(* IEC 61131-3 sources: SmartHomeNew/ (part 10) *)

(* ---- FB_Water_Valve_Runtime_Governance.st ---- *)
FUNCTION_BLOCK FB_Water_Valve_Runtime_Governance
VAR_INPUT
    VI_Enable : BOOL;
    VI_System_Time_MS : UDINT;
END_VAR
VAR
    L_i : INT;
    L_Group : INT;
    L_Feedback_Index_A : INT;
    L_Feedback_Index_B : INT;

    L_Authority : ST_Water_Isolation_Authority_State;
    L_Valve : ST_Water_Valve_Runtime_State;
    L_Empty_Valve : ST_Water_Valve_Runtime_State;

    L_Feedback_A : ST_Water_Valve_Feedback_State;
    L_Feedback_B : ST_Water_Valve_Feedback_State;

    L_Any_Degraded : BOOL;
    L_Any_Confirmation_Unknown : BOOL;
    L_Any_Unsafe_Reopen : BOOL;
END_VAR

IF NOT VI_Enable THEN
    GVL_Water_Valve_Runtime.G_Runtime_Valid := FALSE;
    RETURN;
END_IF;

L_Any_Degraded := FALSE;
L_Any_Confirmation_Unknown := FALSE;
L_Any_Unsafe_Reopen := FALSE;

FOR L_i := 1 TO GVL_CONSTANTS.C_MAX_FLOOD_SENSORS DO

    L_Authority :=
        GVL_Water_Isolation_Authority.G_Authority_State[L_i];

    L_Valve := L_Empty_Valve;
    L_Valve.Runtime_Valid := TRUE;

    L_Valve.Runtime_System_Time_MS := VI_System_Time_MS;

    L_Valve.Valve_Id := L_Authority.Valve_Group_Id;
    L_Valve.Valve_Group_Id := L_Authority.Valve_Group_Id;

    L_Valve.Close_Requested :=
        L_Authority.Selective_Authority_Allowed
        OR L_Authority.Global_Fallback_Required;

    L_Valve.Global_Fallback_Request :=
        L_Authority.Global_Fallback_Required;

    L_Valve.Selective_Authority_Allowed :=
        L_Authority.Selective_Authority_Allowed;

    // Observe-only compatibility visibility.
    L_Valve.Physical_Output_Active :=
        GVL_COMMAND_SHADOW.G_Close_Valve_35
        OR GVL_COMMAND_SHADOW.G_Close_Valve_36;

    L_Valve.Output_Command_Projected :=
        L_Valve.Close_Requested;

    // Feedback/runtime hooks. Runtime authority is per leak sensor, but valve
    // feedback is per physical valve pair: group 1 => 1/2, group 2 => 3/4,
    // group 3 => 5/6, group 4 => 7/8 (35/36).
    L_Group := UINT_TO_INT(L_Authority.Valve_Group_Id);
    L_Feedback_Index_A := 0;
    L_Feedback_Index_B := 0;

    CASE L_Group OF
        1:
            L_Feedback_Index_A := 1;
            L_Feedback_Index_B := 2;
        2:
            L_Feedback_Index_A := 3;
            L_Feedback_Index_B := 4;
        3:
            L_Feedback_Index_A := 5;
            L_Feedback_Index_B := 6;
        4:
            L_Feedback_Index_A := 7;
            L_Feedback_Index_B := 8;
    ELSE
            L_Feedback_Index_A := 0;
            L_Feedback_Index_B := 0;
    END_CASE;

    IF (L_Feedback_Index_A >= 1) AND (L_Feedback_Index_B >= 1) THEN
        L_Feedback_A := GVL_Water_Valve_Feedback.G_Valve_Feedback_State[L_Feedback_Index_A];
        L_Feedback_B := GVL_Water_Valve_Feedback.G_Valve_Feedback_State[L_Feedback_Index_B];

        L_Valve.Confirmation_Available :=
            L_Feedback_A.Feedback_Available
            AND L_Feedback_B.Feedback_Available;

        IF L_Valve.Confirmation_Available THEN
            L_Valve.Confirmed_Closed :=
                L_Feedback_A.Confirmed_Closed
                AND L_Feedback_B.Confirmed_Closed;

            L_Valve.Confirmed_Open :=
                L_Feedback_A.Confirmed_Open
                AND L_Feedback_B.Confirmed_Open;

            L_Valve.Confirmation_Timeout :=
                L_Feedback_A.Feedback_Timeout
                OR L_Feedback_B.Feedback_Timeout;
        ELSE
            L_Valve.Confirmation_Unknown := TRUE;
        END_IF;
    ELSE
        L_Valve.Confirmation_Unknown := TRUE;
    END_IF;

    IF L_Valve.Confirmation_Available
       AND NOT L_Valve.Confirmed_Open
       AND NOT L_Valve.Confirmed_Closed THEN
        L_Valve.Confirmation_Unknown := TRUE;
    END_IF;

    // Observe-only semantics must not force degraded state.
    L_Valve.Diagnostics_Available := FALSE;
    L_Valve.Valve_Healthy := TRUE;

    IF L_Valve.Confirmation_Available
       AND NOT L_Valve.Confirmed_Closed
       AND L_Valve.Close_Requested THEN

        L_Valve.Valve_Degraded := TRUE;

    END_IF;

    IF L_Valve.Confirmation_Timeout THEN
        L_Valve.Valve_Degraded := TRUE;
        L_Valve.Valve_Stuck_Suspected := TRUE;
    END_IF;

    IF L_Valve.Valve_Degraded THEN

        L_Valve.Unsafe_Reopen_Denied := TRUE;
        L_Valve.Recovery_Allowed := FALSE;

        L_Valve.Status_Code := 2;
        L_Valve.Status_Text :=
            'Recovery denied: valve pair degraded';

    ELSIF L_Valve.Confirmation_Unknown THEN

        L_Valve.Status_Code := 1;
        L_Valve.Status_Text :=
            'Valve pair confirmation unavailable';

    ELSE

        L_Valve.Status_Code := 0;
        L_Valve.Status_Text :=
            'Valve pair governance runtime healthy';

    END_IF;

    GVL_Water_Valve_Runtime.G_Valve_Runtime_State[L_i] :=
        L_Valve;

    L_Any_Degraded :=
        L_Any_Degraded
        OR L_Valve.Valve_Degraded;

    L_Any_Confirmation_Unknown :=
        L_Any_Confirmation_Unknown
        OR L_Valve.Confirmation_Unknown;

    L_Any_Unsafe_Reopen :=
        L_Any_Unsafe_Reopen
        OR L_Valve.Unsafe_Reopen_Denied;

END_FOR;

GVL_Water_Valve_Runtime.G_Any_Valve_Degraded :=
    L_Any_Degraded;

GVL_Water_Valve_Runtime.G_Any_Confirmation_Unknown :=
    L_Any_Confirmation_Unknown;

GVL_Water_Valve_Runtime.G_Any_Unsafe_Reopen_Denied :=
    L_Any_Unsafe_Reopen;

GVL_Water_Valve_Runtime.G_Runtime_Valid := TRUE;
GVL_Water_Valve_Runtime.G_Last_Update_MS := VI_System_Time_MS;

IF L_Any_Degraded THEN
    GVL_Water_Valve_Runtime.G_Status_Code := 2;
    GVL_Water_Valve_Runtime.G_Status_Text :=
        'Valve governance degraded';
ELSIF L_Any_Confirmation_Unknown THEN
    GVL_Water_Valve_Runtime.G_Status_Code := 1;
    GVL_Water_Valve_Runtime.G_Status_Text :=
        'Valve pair confirmation unknown';
ELSE
    GVL_Water_Valve_Runtime.G_Status_Code := 0;
    GVL_Water_Valve_Runtime.G_Status_Text :=
        'Valve governance runtime active';
END_IF;

END_FUNCTION_BLOCK

(* ---- FB_Zone_Access_Manager.st ---- *)
FUNCTION_BLOCK FB_Zone_Access_Manager
VAR_INPUT
    VI_System_Time_MS : UDINT; // Системное время (мс)
    VI_Operator_ID    : STRING(10); // Идентификатор оператора
    VI_Target_Zone    : INT; // Номер целевой зоны
    VI_Rights         : ST_Operator_Zone_Rights; // Права доступа оператора к зоне
END_VAR
VAR_OUTPUT
    VO_Access_Granted : BOOL; // Флаг: Доступ разрешен
END_VAR

// Проверка прав доступа к зоне
IF VI_Target_Zone >= 1 AND VI_Target_Zone <= 32 THEN
    // Если глобальный уровень доступа высокий (например, CONFIG или FULL), разрешаем доступ ко всем зонам
    IF VI_Rights.global_access_level >= TO_BYTE(E_Zone_Access_Level.ZONE_ACCESS_CONFIG) THEN
        VO_Access_Granted := TRUE;
    ELSE
        // Иначе проверяем битовую маску для конкретной зоны
        // Бит 0 соответствует зоне 1, бит 1 - зоне 2 и т.д.
        VO_Access_Granted := (VI_Rights.zone_masks AND SHL(DWORD#1, VI_Target_Zone - 1)) <> 0;
    END_IF;
ELSE
    VO_Access_Granted := FALSE;
END_IF;

(* ---- MAIN.st ---- *)
PROGRAM MAIN

// ======================================================
// MAIN CYCLIC EXECUTION PIPELINE
// ======================================================
// Required CODESYS Task Configuration:
//   - Assign only PROGRAM MAIN to the cyclic task.
//   - Do not assign child PRG_* programs directly to the same task.
//   - Configure the real cycle time in CODESYS Task Configuration.
//   - Recommended main control cycle: 100 ms.
// ======================================================

// 1. Time / init / configuration
PRG_Time_Service();
PRG_Time_Monotonic_Governor();
PRG_System_Init();
PRG_Config_Manager();
PRG_Config_Validation();
PRG_Config_Versioning();
PRG_System_Runtime_Base();

// 2. Peer heartbeat ingestion
PRG_Peer_Heartbeat_Ingestion();

// 3. PLC role arbitration
PRG_PLC_Arbitration();

// 4. PLC ownership / fencing governance
PRG_PLC_Fencing_Governor();

// 5. IO read, passive quality observation and normalized inputs
PRG_IO_Read();
PRG_Input_Quality_Read();
PRG_Input_Processing();

// 6. Base mode, presence and safety
PRG_Mode_Manager();
PRG_Presence_Manager();
PRG_Safety();
PRG_Safety_Operator();
PRG_Safety_Shutdown();
PRG_Safety_Recovery();

// 7. Intent, adaptive behavior, scenario and policy
PRG_System_Intent();
PRG_Security();
PRG_System_Access_Maintenance();
PRG_User_Adapt_Control();
PRG_Behavior_Adapt_Profile();
PRG_Scenario_Engine();
PRG_System_Scenario_Rules();
PRG_System_Evacuation();
PRG_Policy();
PRG_Heating_Policy_Manager();
PRG_Heating_Policy_Observer();
PRG_System_Coordinator();

// 8. Command arbitration
PRG_Command_Arbitration();

// 9. Transport pipeline
PRG_Modbus_Master();
PRG_Modbus_RTU_Bridge();
PRG_Modbus_RTU_Driver();
PRG_Modbus_RTU_SysCom_Backend();
PRG_Modbus_RTU_SysCom_Transport();
PRG_Modbus_Register_Scan();
PRG_OpenTherm_Transport();
PRG_OpenTherm_Adapter_Status();

// 10. Transport freshness governance
PRG_Transport_Freshness_Governor();

// 11. Runtime authority barrier
PRG_Runtime_Barrier();

// 12. Immutable runtime snapshot governance
PRG_Runtime_Snapshot_Governor();

// 13. Canonical peer session publication
PRG_Peer_Session_Publication();

// 14. HA session replication boundary
PRG_HA_Session_Replication();

// 15. Distributed peer ingestion
PRG_Distributed_Peer_Ingestion();

// 16. Distributed epoch reconciliation governance
PRG_Distributed_Epoch_Governor();

// 17. Distributed snapshot publication
PRG_Distributed_Snapshot_Publication();

// 18. Distributed snapshot ingestion
PRG_Distributed_Snapshot_Ingestion();

// 19. Distributed immutable snapshot reconciliation governance
PRG_Distributed_Snapshot_Governor();

// 20. Distributed runtime fabric supervisor
PRG_Distributed_Runtime_Supervisor();

// 21. Distributed commit publication
PRG_Distributed_Commit_Publication();

// 22. Distributed commit ingestion
PRG_Distributed_Commit_Ingestion();

// 23. Distributed deterministic publication commit governance
PRG_Distributed_Commit_Governor();

// 24. Distributed deterministic commit observability projection
PRG_Distributed_Commit_Observability();

// 25. Semantic execution continuity governance
PRG_Semantic_Progress_Governor();

// 26. Systemic convergence governance
PRG_Convergence_Governor();

// 27. Recovery cleanup governance
PRG_Recovery_Cleanup_Governor();

// 28. Observability authority governance
PRG_Observability_Governor();

// 29. Domain execution and projection
PRG_Heating();
PRG_Heating_Supervisory_Publication();
PRG_Ventilation();
PRG_Water_Supervisory_Publication();
PRG_Water_Output_Projection();
PRG_Water();
PRG_Access();
PRG_Lighting();

// 30. Output freshness governance
PRG_Output_Freshness_Governor();

// 31. Immutable physical snapshot governance
PRG_Physical_Snapshot_Governor();

// 32. Physical sensor consensus governance
PRG_Sensor_Consensus_Governor();

// 33. Telemetry causality governance
PRG_Telemetry_Causality_Governor();

// 34. Global physical authority epoch governance
PRG_Physical_Authority_Epoch_Governor();

// 35. Persistent authority lineage governance
PRG_Authority_Lineage_Governor();

// 36. Global authority revocation governance
PRG_Authority_Revocation_Governor();

// 37. Deterministic authority restoration governance
PRG_Authority_Restoration_Governor();

// 38. Pre-output safety barrier
PRG_PreOutput_Safety_Barrier();

// 39. Final physical IO projection
PRG_IO_Write();

// 40. Deterministic field actuation governance
PRG_Actuation_Authority_Governor();

// 41. Deterministic physical transaction governance
PRG_Physical_Transaction_Governor();

// 42. Deterministic temporal stability governance
PRG_Temporal_Stability_Governor();

// 43. Environmental authority governance
PRG_Environmental_Authority_Governor();

// 44. Runtime resource authority governance
PRG_Runtime_Resource_Authority_Governor();

// 45. Semantic continuity authority governance
PRG_Semantic_Continuity_Authority_Governor();

// 46. Authoritative observability truth governance
PRG_Observability_Truth_Governor();

// 47. Immutable historical truth governance
PRG_Historical_Truth_Governor();

// 48. Global synchronized authority governance
PRG_Global_Authority_Sync_Governor();

// 49. Deterministic control temporal coherence governance
PRG_Control_Temporal_Coherence_Governor();

// 50. Physical actuator semantic verification governance
PRG_Actuator_Semantic_Verification_Governor();

// 51. Deterministic energy causality governance
PRG_Energy_Causality_Governor();

// 52. Deterministic runtime sustainability governance
PRG_Runtime_Sustainability_Governor();

// 53. Deterministic semantic preservation governance
PRG_Semantic_Preservation_Governor();

// 54. Deterministic operator semantic alignment governance
PRG_Operator_Semantic_Alignment_Governor();

// 55. Deterministic ecosystem semantic federation governance
PRG_Semantic_Federation_Governor();

// 56. Deterministic compliance federation governance
PRG_Compliance_Federation_Governor();

// 57. Deterministic forensic evidence governance
PRG_Forensic_Evidence_Governor();

// 58. Deterministic epistemic integrity governance
PRG_Epistemic_Integrity_Governor();

// 59. Deterministic meta-governance consistency governance
// Must run before observability authority publication to guarantee
// acyclic and independently grounded governance topology.
PRG_Meta_Governance_Governor();

// 60. Observability authority coherence governance
PRG_Observability_Authority_Governor();

// 61. Verification, diagnostics, history, HMI
PRG_Command_Verifier();
PRG_Explainability();
PRG_System_Health();
PRG_System_Alarm_Gateway();
PRG_System_Diagnostics();
PRG_System_Diagnostics_Ext();
PRG_System_History();
PRG_System_BlackBox();
PRG_System_Trend();
PRG_System_Simulation();
PRG_HMI_Dashboard();
PRG_Debug_View();

// >>> BULK_SYNC_ANCHOR: MAIN <<<
END_PROGRAM

(* ---- PRG_Access.st ---- *)
PROGRAM PRG_Access
VAR
    fbProjection : FB_Access_Output_Projection;

    fbPulseLock1Open : FB_Access_Pulse_Channel;
    fbPulseLock1Close : FB_Access_Pulse_Channel;
    fbPulseLock2Open : FB_Access_Pulse_Channel;
    fbPulseLock2Close : FB_Access_Pulse_Channel;
    fbPulseGateOpen : FB_Access_Pulse_Channel;
    fbPulseWicketOpen : FB_Access_Pulse_Channel;

    L_Mode : E_Safety_Mode;
    L_Now_MS : UDINT;
    L_Pulse_MS : UDINT;

    L_Distributed_Execute_Allowed : BOOL;
    L_Distributed_Access_Allowed : BOOL;

    L_Lock_1_Open : BOOL;
    L_Lock_1_Close : BOOL;
    L_Lock_2_Open : BOOL;
    L_Lock_2_Close : BOOL;
    L_Gate_Open : BOOL;
    L_Wicket_Open : BOOL;
END_VAR

L_Mode := GVL_SAFETY_SHUTDOWN.G_Safety_Mode;
L_Now_MS := GVL_STATUS.G_System_Time_MS;

GVL_ACCESS_RUNTIME.G_Runtime_Required := FALSE;
GVL_ACCESS_RUNTIME.G_Runtime_Executed := TRUE;
GVL_ACCESS_RUNTIME.G_Runtime_Idle_By_Design := FALSE;
GVL_ACCESS_RUNTIME.G_Runtime_Blocked_By_Distributed_Gates := FALSE;
GVL_ACCESS_RUNTIME.G_Any_Pulse_Active := FALSE;
GVL_ACCESS_RUNTIME.G_Last_Update_MS := L_Now_MS;

// Distributed runtime governance.
// FIRE/GAS emergency semantics remain authoritative.
L_Distributed_Execute_Allowed :=
    GVL_Distributed_Execution_Gates.G_Can_Execute;

L_Distributed_Access_Allowed :=
    GVL_Distributed_Execution_Gates.G_Can_Own_Projection;

IF (L_Mode <> FIRE)
   AND (L_Mode <> GAS)
   AND (
        NOT L_Distributed_Execute_Allowed
        OR NOT L_Distributed_Access_Allowed
       ) THEN

    // Clear all pulse channels before blocking projection to avoid stale pulse-active state.
    fbPulseLock1Open(VI_Command := FALSE, VI_Reset := TRUE, VI_Now_MS := L_Now_MS, VI_Pulse_MS := 100);
    fbPulseLock1Close(VI_Command := FALSE, VI_Reset := TRUE, VI_Now_MS := L_Now_MS, VI_Pulse_MS := 100);
    fbPulseLock2Open(VI_Command := FALSE, VI_Reset := TRUE, VI_Now_MS := L_Now_MS, VI_Pulse_MS := 100);
    fbPulseLock2Close(VI_Command := FALSE, VI_Reset := TRUE, VI_Now_MS := L_Now_MS, VI_Pulse_MS := 100);
    fbPulseGateOpen(VI_Command := FALSE, VI_Reset := TRUE, VI_Now_MS := L_Now_MS, VI_Pulse_MS := 100);
    fbPulseWicketOpen(VI_Command := FALSE, VI_Reset := TRUE, VI_Now_MS := L_Now_MS, VI_Pulse_MS := 100);

    fbProjection(
        VI_Lock_1_Open := FALSE,
        VI_Lock_1_Close := FALSE,
        VI_Lock_2_Open := FALSE,
        VI_Lock_2_Close := FALSE,
        VI_Gate_Open := FALSE,
        VI_Wicket_Open := FALSE
    );

    GVL_ACCESS_RUNTIME.G_Runtime_Blocked_By_Distributed_Gates := TRUE;
    GVL_ACCESS_RUNTIME.G_Any_Pulse_Active := FALSE;
    GVL_ACCESS_RUNTIME.G_Status_Code := 2;
    GVL_ACCESS_RUNTIME.G_Status_Text := 'Access runtime blocked by distributed gates';

    RETURN;
END_IF;

// Access is not part of WATER_LEAK or GLOBAL_STOP recovery semantics.
// Clear active one-shot pulses so old manual commands cannot continue during safety stop.
IF (L_Mode = WATER_LEAK) OR (L_Mode = GLOBAL_STOP) THEN
    fbPulseLock1Open(VI_Command := FALSE, VI_Reset := TRUE, VI_Now_MS := L_Now_MS, VI_Pulse_MS := 100);
    fbPulseLock1Close(VI_Command := FALSE, VI_Reset := TRUE, VI_Now_MS := L_Now_MS, VI_Pulse_MS := 100);
    fbPulseLock2Open(VI_Command := FALSE, VI_Reset := TRUE, VI_Now_MS := L_Now_MS, VI_Pulse_MS := 100);
    fbPulseLock2Close(VI_Command := FALSE, VI_Reset := TRUE, VI_Now_MS := L_Now_MS, VI_Pulse_MS := 100);
    fbPulseGateOpen(VI_Command := FALSE, VI_Reset := TRUE, VI_Now_MS := L_Now_MS, VI_Pulse_MS := 100);
    fbPulseWicketOpen(VI_Command := FALSE, VI_Reset := TRUE, VI_Now_MS := L_Now_MS, VI_Pulse_MS := 100);

    fbProjection(
        VI_Lock_1_Open := FALSE,
        VI_Lock_1_Close := FALSE,
        VI_Lock_2_Open := FALSE,
        VI_Lock_2_Close := FALSE,
        VI_Gate_Open := FALSE,
        VI_Wicket_Open := FALSE
    );

    GVL_ACCESS_RUNTIME.G_Runtime_Required := FALSE;
    GVL_ACCESS_RUNTIME.G_Runtime_Idle_By_Design := TRUE;
    GVL_ACCESS_RUNTIME.G_Any_Pulse_Active := FALSE;
    GVL_ACCESS_RUNTIME.G_Status_Code := 3;
    GVL_ACCESS_RUNTIME.G_Status_Text := 'Access runtime safety-cleared';

    RETURN;
END_IF;

// Load pulse duration from config with safety clamp.
L_Pulse_MS := GVL_CONFIG.G_Access_Pulse_MS;
IF L_Pulse_MS < 100 THEN
    L_Pulse_MS := 100;
ELSIF L_Pulse_MS > 5000 THEN
    L_Pulse_MS := 5000;
END_IF;

L_Lock_1_Open := FALSE;
L_Lock_1_Close := FALSE;
L_Lock_2_Open := FALSE;
L_Lock_2_Close := FALSE;
L_Gate_Open := FALSE;
L_Wicket_Open := FALSE;

CASE L_Mode OF
    FIRE:
        // Fire evacuation access commands are authoritative and continuous.
        L_Lock_1_Open := GVL_COMMAND_SHADOW.G_Lock_1_Open;
        L_Lock_2_Open := GVL_COMMAND_SHADOW.G_Lock_2_Open;
        L_Gate_Open := GVL_COMMAND_SHADOW.G_Gate_Open;
        L_Wicket_Open := GVL_COMMAND_SHADOW.G_Wicket_Open;

        // Synchronize pulse channels with current command state and clear active pulses.
        fbPulseLock1Open(VI_Command := GVL_COMMAND_SHADOW.G_Lock_1_Open, VI_Reset := TRUE, VI_Now_MS := L_Now_MS, VI_Pulse_MS := L_Pulse_MS);
        fbPulseLock1Close(VI_Command := GVL_COMMAND_SHADOW.G_Lock_1_Close, VI_Reset := TRUE, VI_Now_MS := L_Now_MS, VI_Pulse_MS := L_Pulse_MS);
        fbPulseLock2Open(VI_Command := GVL_COMMAND_SHADOW.G_Lock_2_Open, VI_Reset := TRUE, VI_Now_MS := L_Now_MS, VI_Pulse_MS := L_Pulse_MS);
        fbPulseLock2Close(VI_Command := GVL_COMMAND_SHADOW.G_Lock_2_Close, VI_Reset := TRUE, VI_Now_MS := L_Now_MS, VI_Pulse_MS := L_Pulse_MS);
        fbPulseGateOpen(VI_Command := GVL_COMMAND_SHADOW.G_Gate_Open, VI_Reset := TRUE, VI_Now_MS := L_Now_MS, VI_Pulse_MS := L_Pulse_MS);
        fbPulseWicketOpen(VI_Command := GVL_COMMAND_SHADOW.G_Wicket_Open, VI_Reset := TRUE, VI_Now_MS := L_Now_MS, VI_Pulse_MS := L_Pulse_MS);

    GAS:
        // Gas mode uses direct gate opening plus limited pulsed pedestrian/lock release.
        L_Gate_Open := GVL_COMMAND_SHADOW.G_Gate_Open;

        fbPulseLock1Open(VI_Command := GVL_COMMAND_SHADOW.G_Lock_1_Open, VI_Reset := FALSE, VI_Now_MS := L_Now_MS, VI_Pulse_MS := L_Pulse_MS);
        fbPulseLock2Open(VI_Command := GVL_COMMAND_SHADOW.G_Lock_2_Open, VI_Reset := FALSE, VI_Now_MS := L_Now_MS, VI_Pulse_MS := L_Pulse_MS);
        fbPulseWicketOpen(VI_Command := GVL_COMMAND_SHADOW.G_Wicket_Open, VI_Reset := FALSE, VI_Now_MS := L_Now_MS, VI_Pulse_MS := L_Pulse_MS);

        fbPulseLock1Close(VI_Command := GVL_COMMAND_SHADOW.G_Lock_1_Close, VI_Reset := TRUE, VI_Now_MS := L_Now_MS, VI_Pulse_MS := L_Pulse_MS);
        fbPulseLock2Close(VI_Command := GVL_COMMAND_SHADOW.G_Lock_2_Close, VI_Reset := TRUE, VI_Now_MS := L_Now_MS, VI_Pulse_MS := L_Pulse_MS);
        fbPulseGateOpen(VI_Command := GVL_COMMAND_SHADOW.G_Gate_Open, VI_Reset := TRUE, VI_Now_MS := L_Now_MS, VI_Pulse_MS := L_Pulse_MS);

        L_Lock_1_Open := fbPulseLock1Open.VO_Output;
        L_Lock_2_Open := fbPulseLock2Open.VO_Output;
        L_Wicket_Open := fbPulseWicketOpen.VO_Output;

ELSE
        fbPulseLock1Open(VI_Command := GVL_COMMAND_SHADOW.G_Lock_1_Open, VI_Reset := FALSE, VI_Now_MS := L_Now_MS, VI_Pulse_MS := L_Pulse_MS);
        fbPulseLock1Close(VI_Command := GVL_COMMAND_SHADOW.G_Lock_1_Close, VI_Reset := FALSE, VI_Now_MS := L_Now_MS, VI_Pulse_MS := L_Pulse_MS);
        fbPulseLock2Open(VI_Command := GVL_COMMAND_SHADOW.G_Lock_2_Open, VI_Reset := FALSE, VI_Now_MS := L_Now_MS, VI_Pulse_MS := L_Pulse_MS);
        fbPulseLock2Close(VI_Command := GVL_COMMAND_SHADOW.G_Lock_2_Close, VI_Reset := FALSE, VI_Now_MS := L_Now_MS, VI_Pulse_MS := L_Pulse_MS);
        fbPulseGateOpen(VI_Command := GVL_COMMAND_SHADOW.G_Gate_Open, VI_Reset := FALSE, VI_Now_MS := L_Now_MS, VI_Pulse_MS := L_Pulse_MS);
        fbPulseWicketOpen(VI_Command := GVL_COMMAND_SHADOW.G_Wicket_Open, VI_Reset := FALSE, VI_Now_MS := L_Now_MS, VI_Pulse_MS := L_Pulse_MS);

        L_Lock_1_Open := fbPulseLock1Open.VO_Output;
        L_Lock_1_Close := fbPulseLock1Close.VO_Output;
        L_Lock_2_Open := fbPulseLock2Open.VO_Output;
        L_Lock_2_Close := fbPulseLock2Close.VO_Output;
        L_Gate_Open := fbPulseGateOpen.VO_Output;
        L_Wicket_Open := fbPulseWicketOpen.VO_Output;
END_CASE;

GVL_ACCESS_RUNTIME.G_Any_Pulse_Active :=
    fbPulseLock1Open.VO_Active
    OR fbPulseLock1Close.VO_Active
    OR fbPulseLock2Open.VO_Active
    OR fbPulseLock2Close.VO_Active
    OR fbPulseGateOpen.VO_Active
    OR fbPulseWicketOpen.VO_Active;

GVL_ACCESS_RUNTIME.G_Runtime_Required :=
    (L_Mode = FIRE)
    OR (L_Mode = GAS)
    OR GVL_COMMAND_SHADOW.G_Lock_1_Open
    OR GVL_COMMAND_SHADOW.G_Lock_1_Close
    OR GVL_COMMAND_SHADOW.G_Lock_2_Open
    OR GVL_COMMAND_SHADOW.G_Lock_2_Close
    OR GVL_COMMAND_SHADOW.G_Gate_Open
    OR GVL_COMMAND_SHADOW.G_Wicket_Open
    OR GVL_ACCESS_RUNTIME.G_Any_Pulse_Active;

GVL_ACCESS_RUNTIME.G_Runtime_Idle_By_Design :=
    NOT GVL_ACCESS_RUNTIME.G_Runtime_Required;

IF GVL_ACCESS_RUNTIME.G_Runtime_Idle_By_Design THEN
    GVL_ACCESS_RUNTIME.G_Status_Code := 0;
    GVL_ACCESS_RUNTIME.G_Status_Text := 'Access runtime idle by design';
ELSE
    GVL_ACCESS_RUNTIME.G_Status_Code := 1;
    GVL_ACCESS_RUNTIME.G_Status_Text := 'Access runtime active';
END_IF;

fbProjection(
    VI_Lock_1_Open := L_Lock_1_Open,
    VI_Lock_1_Close := L_Lock_1_Close,
    VI_Lock_2_Open := L_Lock_2_Open,
    VI_Lock_2_Close := L_Lock_2_Close,
    VI_Gate_Open := L_Gate_Open,
    VI_Wicket_Open := L_Wicket_Open
);

// >>> BULK_SYNC_ANCHOR: PRG_Access <<<
END_PROGRAM

(* ---- PRG_Actuation_Authority_Governor.st ---- *)
PROGRAM PRG_Actuation_Authority_Governor
VAR
    L_Now_MS : UDINT;
    L_Actuation_Valid : BOOL := TRUE;
    L_Error_Code : UDINT := 0;
    L_Error_Text : STRING(160) := '';
END_VAR

L_Now_MS := GVL_STATUS.G_System_Time_MS;
L_Actuation_Valid := TRUE;
L_Error_Code := 0;
L_Error_Text := '';

GVL_ACTUATION_AUTHORITY.Actuation_Authority_Valid := FALSE;
GVL_ACTUATION_AUTHORITY.Actuation_Authority_Granted := FALSE;
GVL_ACTUATION_AUTHORITY.Actuation_Quarantine_Active := TRUE;
GVL_ACTUATION_AUTHORITY.Field_Device_ACK_Valid := FALSE;
GVL_ACTUATION_AUTHORITY.Actuator_Transition_Observed := FALSE;
GVL_ACTUATION_AUTHORITY.Physical_Convergence_Confirmed := FALSE;
GVL_ACTUATION_AUTHORITY.Stable_Physical_Convergence := FALSE;

GVL_ACTUATION_AUTHORITY.Actuation_Command_Epoch := ULINT_TO_UDINT(GVL_OUTPUT_EPOCH.Output_Publication_Epoch);

IF GVL_ACTUATION_AUTHORITY.Field_ACK_Epoch <> GVL_ACTUATION_AUTHORITY.Actuation_Command_Epoch THEN
    GVL_ACTUATION_AUTHORITY.Command_Actuation_Skew_Detected := TRUE;
    L_Actuation_Valid := FALSE;
    L_Error_Code := 26000;
    L_Error_Text := 'Command actuation epoch skew detected';
END_IF;

IF L_Actuation_Valid AND GVL_ACTUATION_AUTHORITY.ACK_Replay_Suspected THEN
    L_Actuation_Valid := FALSE;
    L_Error_Code := 26001;
    L_Error_Text := 'Field ACK replay suspected';
END_IF;

IF L_Actuation_Valid AND GVL_ACTUATION_AUTHORITY.Write_Without_Confirm_Detected THEN
    L_Actuation_Valid := FALSE;
    L_Error_Code := 26002;
    L_Error_Text := 'Write without field confirmation detected';
END_IF;

IF L_Actuation_Valid AND GVL_ACTUATION_AUTHORITY.Relay_Weld_Suspected THEN
    L_Actuation_Valid := FALSE;
    L_Error_Code := 26003;
    L_Error_Text := 'Relay weld suspected';
END_IF;

IF L_Actuation_Valid AND GVL_ACTUATION_AUTHORITY.Actuator_Stall_Detected THEN
    L_Actuation_Valid := FALSE;
    L_Error_Code := 26004;
    L_Error_Text := 'Actuator stall detected';
END_IF;

IF L_Actuation_Valid AND GVL_ACTUATION_AUTHORITY.Partial_Actuation_Detected THEN
    L_Actuation_Valid := FALSE;
    L_Error_Code := 26005;
    L_Error_Text := 'Partial actuation detected';
END_IF;

IF L_Actuation_Valid AND NOT GVL_ACTUATION_AUTHORITY.Current_Signature_Confirmed THEN
    L_Actuation_Valid := FALSE;
    L_Error_Code := 26010;
    L_Error_Text := 'Current signature confirmation missing';
END_IF;

IF L_Actuation_Valid AND NOT GVL_ACTUATION_AUTHORITY.Flow_Response_Confirmed THEN
    L_Actuation_Valid := FALSE;
    L_Error_Code := 26011;
    L_Error_Text := 'Flow response confirmation missing';
END_IF;

IF L_Actuation_Valid AND NOT GVL_ACTUATION_AUTHORITY.Pressure_Response_Confirmed THEN
    L_Actuation_Valid := FALSE;
    L_Error_Code := 26012;
    L_Error_Text := 'Pressure response confirmation missing';
END_IF;

IF L_Actuation_Valid AND NOT GVL_ACTUATION_AUTHORITY.Motion_Response_Confirmed THEN
    L_Actuation_Valid := FALSE;
    L_Error_Code := 26013;
    L_Error_Text := 'Motion response confirmation missing';
END_IF;

IF L_Actuation_Valid THEN
    GVL_ACTUATION_AUTHORITY.Actuation_Authority_Valid := TRUE;
    GVL_ACTUATION_AUTHORITY.Actuation_Authority_Granted := TRUE;
    GVL_ACTUATION_AUTHORITY.Actuation_Quarantine_Active := FALSE;
    GVL_ACTUATION_AUTHORITY.Field_Device_ACK_Valid := TRUE;
    GVL_ACTUATION_AUTHORITY.Actuator_Transition_Observed := TRUE;
    GVL_ACTUATION_AUTHORITY.Physical_Convergence_Confirmed := TRUE;
    GVL_ACTUATION_AUTHORITY.Stable_Physical_Convergence := TRUE;
    GVL_ACTUATION_AUTHORITY.Actuation_Authority_Epoch := GVL_ACTUATION_AUTHORITY.Actuation_Command_Epoch;
    GVL_ACTUATION_AUTHORITY.Actuation_Last_Update_MS := L_Now_MS;
    GVL_ACTUATION_AUTHORITY.Actuation_Lease_Expired := FALSE;
    GVL_ACTUATION_AUTHORITY.Actuation_Last_Error_Code := 0;
    GVL_ACTUATION_AUTHORITY.Actuation_Last_Error_Text := '';
ELSE
    GVL_ACTUATION_AUTHORITY.Actuation_Authority_Valid := FALSE;
    GVL_ACTUATION_AUTHORITY.Actuation_Authority_Granted := FALSE;
    GVL_ACTUATION_AUTHORITY.Actuation_Quarantine_Active := TRUE;
    GVL_ACTUATION_AUTHORITY.Actuation_Lease_Expired := TRUE;
    GVL_ACTUATION_AUTHORITY.Actuation_Last_Error_Code := L_Error_Code;
    GVL_ACTUATION_AUTHORITY.Actuation_Last_Error_Text := L_Error_Text;
    GVL_ACTUATION_AUTHORITY.Actuation_Invalidation_Count := GVL_ACTUATION_AUTHORITY.Actuation_Invalidation_Count + 1;
END_IF;

END_PROGRAM

(* ---- PRG_Actuator_Semantic_Verification_Governor.st ---- *)
PROGRAM PRG_Actuator_Semantic_Verification_Governor
VAR
    L_Now_MS : UDINT;
    L_Actuator_Valid : BOOL := TRUE;
    L_Error_Code : UDINT := 0;
    L_Error_Text : STRING(160) := '';
END_VAR

L_Now_MS := GVL_STATUS.G_System_Time_MS;
L_Actuator_Valid := TRUE;
L_Error_Code := 0;
L_Error_Text := '';

// Fail-safe defaults.
GVL_ACTUATOR_SEMANTIC_VERIFICATION.Actuator_Semantic_Verification_Valid := FALSE;
GVL_ACTUATOR_SEMANTIC_VERIFICATION.Actuator_Semantic_Verification_Granted := FALSE;
GVL_ACTUATOR_SEMANTIC_VERIFICATION.Actuator_Semantic_Verification_Quarantine_Active := TRUE;

GVL_ACTUATOR_SEMANTIC_VERIFICATION.Valve_Semantic_Realization_Valid := FALSE;
GVL_ACTUATOR_SEMANTIC_VERIFICATION.Relay_Semantic_Realization_Valid := FALSE;
GVL_ACTUATOR_SEMANTIC_VERIFICATION.Pump_Semantic_Realization_Valid := FALSE;
GVL_ACTUATOR_SEMANTIC_VERIFICATION.Fan_Semantic_Realization_Valid := FALSE;
GVL_ACTUATOR_SEMANTIC_VERIFICATION.Hydraulic_Response_Valid := FALSE;

// Control temporal coherence required.
IF NOT GVL_CONTROL_TIMING_FABRIC.Control_Temporal_Coherence_Granted THEN
    L_Actuator_Valid := FALSE;
    L_Error_Code := 36000;
    L_Error_Text := 'Control temporal coherence not granted';
END_IF;

// Semantic realization failure detectors.
IF GVL_ACTUATOR_SEMANTIC_VERIFICATION.False_Positive_Actuation_Detected THEN
    L_Actuator_Valid := FALSE;
    L_Error_Code := 36001;
    L_Error_Text := 'False-positive actuation detected';
END_IF;

IF GVL_ACTUATOR_SEMANTIC_VERIFICATION.Mechanical_NonRealization_Detected THEN
    L_Actuator_Valid := FALSE;
    L_Error_Code := 36002;
    L_Error_Text := 'Mechanical non-realization detected';
END_IF;

IF GVL_ACTUATOR_SEMANTIC_VERIFICATION.Welded_Relay_Semantics_Detected THEN
    L_Actuator_Valid := FALSE;
    L_Error_Code := 36003;
    L_Error_Text := 'Welded relay semantics detected';
END_IF;

IF GVL_ACTUATOR_SEMANTIC_VERIFICATION.Hydraulic_NoEffect_Execution_Detected THEN
    L_Actuator_Valid := FALSE;
    L_Error_Code := 36004;
    L_Error_Text := 'Hydraulic no-effect execution detected';
END_IF;

IF GVL_ACTUATOR_SEMANTIC_VERIFICATION.Airflow_Realization_Mismatch_Detected THEN
    L_Actuator_Valid := FALSE;
    L_Error_Code := 36005;
    L_Error_Text := 'Airflow realization mismatch detected';
END_IF;

IF GVL_ACTUATOR_SEMANTIC_VERIFICATION.Physical_Convergence_Divergence_Detected THEN
    L_Actuator_Valid := FALSE;
    L_Error_Code := 36006;
    L_Error_Text := 'Physical convergence divergence detected';
END_IF;

// Physical semantic convergence validation.
IF L_Actuator_Valid
AND NOT GVL_ACTUATOR_SEMANTIC_VERIFICATION.Physical_Effect_Converged THEN
    L_Actuator_Valid := FALSE;
    L_Error_Code := 36010;
    L_Error_Text := 'Physical effect convergence invalid';
END_IF;

IF L_Actuator_Valid
AND NOT GVL_ACTUATOR_SEMANTIC_VERIFICATION.Actuation_Response_Temporal_Valid THEN
    L_Actuator_Valid := FALSE;
    L_Error_Code := 36011;
    L_Error_Text := 'Actuation response timing invalid';
END_IF;

IF L_Actuator_Valid
AND NOT GVL_ACTUATOR_SEMANTIC_VERIFICATION.Sensor_Confirmed_Execution_Valid THEN
    L_Actuator_Valid := FALSE;
    L_Error_Code := 36012;
    L_Error_Text := 'Sensor-confirmed execution invalid';
END_IF;

IF L_Actuator_Valid
AND NOT GVL_ACTUATOR_SEMANTIC_VERIFICATION.Semantic_Outcome_Aligned THEN
    L_Actuator_Valid := FALSE;
    L_Error_Code := 36013;
    L_Error_Text := 'Semantic outcome alignment invalid';
END_IF;

IF L_Actuator_Valid THEN
    GVL_ACTUATOR_SEMANTIC_VERIFICATION.Actuator_Semantic_Verification_Valid := TRUE;
    GVL_ACTUATOR_SEMANTIC_VERIFICATION.Actuator_Semantic_Verification_Granted := TRUE;
    GVL_ACTUATOR_SEMANTIC_VERIFICATION.Actuator_Semantic_Verification_Quarantine_Active := FALSE;

    GVL_ACTUATOR_SEMANTIC_VERIFICATION.Valve_Semantic_Realization_Valid := TRUE;
    GVL_ACTUATOR_SEMANTIC_VERIFICATION.Relay_Semantic_Realization_Valid := TRUE;
    GVL_ACTUATOR_SEMANTIC_VERIFICATION.Pump_Semantic_Realization_Valid := TRUE;
    GVL_ACTUATOR_SEMANTIC_VERIFICATION.Fan_Semantic_Realization_Valid := TRUE;
    GVL_ACTUATOR_SEMANTIC_VERIFICATION.Hydraulic_Response_Valid := TRUE;

    GVL_ACTUATOR_SEMANTIC_VERIFICATION.Actuator_Verification_Epoch :=
        GVL_CONTROL_TIMING_FABRIC.Control_Timing_Epoch;

    GVL_ACTUATOR_SEMANTIC_VERIFICATION.Actuator_Verification_Epoch_Coherent := TRUE;

    GVL_ACTUATOR_SEMANTIC_VERIFICATION.Actuator_Verification_Last_Update_MS :=
        L_Now_MS;

    GVL_ACTUATOR_SEMANTIC_VERIFICATION.Actuator_Verification_Lease_Expired := FALSE;

    GVL_ACTUATOR_SEMANTIC_VERIFICATION.Actuator_Verification_Last_Error_Code := 0;
    GVL_ACTUATOR_SEMANTIC_VERIFICATION.Actuator_Verification_Last_Error_Text := '';
ELSE
    GVL_ACTUATOR_SEMANTIC_VERIFICATION.Actuator_Semantic_Verification_Valid := FALSE;
    GVL_ACTUATOR_SEMANTIC_VERIFICATION.Actuator_Semantic_Verification_Granted := FALSE;
    GVL_ACTUATOR_SEMANTIC_VERIFICATION.Actuator_Semantic_Verification_Quarantine_Active := TRUE;

    GVL_ACTUATOR_SEMANTIC_VERIFICATION.Actuator_Verification_Lease_Expired := TRUE;

    GVL_ACTUATOR_SEMANTIC_VERIFICATION.Actuator_Verification_Last_Error_Code :=
        L_Error_Code;

    GVL_ACTUATOR_SEMANTIC_VERIFICATION.Actuator_Verification_Last_Error_Text :=
        L_Error_Text;

    GVL_ACTUATOR_SEMANTIC_VERIFICATION.Actuator_Verification_Invalidation_Count :=
        GVL_ACTUATOR_SEMANTIC_VERIFICATION.Actuator_Verification_Invalidation_Count + 1;
END_IF;

END_PROGRAM

(* ---- PRG_Alarm_Audible_Ack_Manager.st ---- *)
PROGRAM PRG_Alarm_Audible_Ack_Manager
VAR
    L_Audible_Alarm_Active : BOOL;
    L_Remaining_MS : UDINT;
END_VAR

L_Audible_Alarm_Active := GVL_ALARM.G_Global_Critical OR GVL_ALARM.G_Gas_Fire_Siren OR GVL_ALARM.G_Security_Siren;
GVL_ALARM_AUDIBLE_ACK.G_Last_Ack_Accepted := FALSE;
GVL_ALARM_AUDIBLE_ACK.G_Last_Ack_Denied := FALSE;
GVL_ALARM_AUDIBLE_ACK.G_Last_Denial_Code := 0;

IF NOT L_Audible_Alarm_Active THEN
    GVL_ALARM_AUDIBLE_ACK.G_Ack_Active := FALSE;
    GVL_ALARM_AUDIBLE_ACK.G_Ack_Expires_MS := 0;
    GVL_ALARM_AUDIBLE_ACK.G_Ack_Remaining_MS := 0;
    GVL_ALARM_AUDIBLE_ACK.G_Ack_Count_Current_Alarm := 0;
    GVL_ALARM_AUDIBLE_ACK.G_Ack_Limit_Reached := FALSE;
    GVL_ALARM_AUDIBLE_ACK.G_Status_Text := 'Audible alarm acknowledgement idle';
END_IF;

IF GVL_ALARM_AUDIBLE_ACK.G_Ack_Active THEN
    IF GVL_TIME_SERVICE.G_Now_MS >= GVL_ALARM_AUDIBLE_ACK.G_Ack_Expires_MS THEN
        GVL_ALARM_AUDIBLE_ACK.G_Ack_Active := FALSE;
        GVL_ALARM_AUDIBLE_ACK.G_Ack_Remaining_MS := 0;
        GVL_ALARM_AUDIBLE_ACK.G_Status_Text := 'Audible alarm acknowledgement expired';
    ELSE
        L_Remaining_MS := GVL_ALARM_AUDIBLE_ACK.G_Ack_Expires_MS - GVL_TIME_SERVICE.G_Now_MS;
        GVL_ALARM_AUDIBLE_ACK.G_Ack_Remaining_MS := L_Remaining_MS;
    END_IF;
END_IF;

IF GVL_ALARM_AUDIBLE_ACK.G_Ack_Request THEN
    IF NOT L_Audible_Alarm_Active THEN
        GVL_ALARM_AUDIBLE_ACK.G_Last_Ack_Denied := TRUE;
        GVL_ALARM_AUDIBLE_ACK.G_Last_Denial_Code := 1;
        GVL_ALARM_AUDIBLE_ACK.G_Status_Text := 'Audible acknowledgement denied: no active audible alarm';
    ELSIF GVL_INTENT_USER.I_User_Access_Level < 2 THEN
        GVL_ALARM_AUDIBLE_ACK.G_Last_Ack_Denied := TRUE;
        GVL_ALARM_AUDIBLE_ACK.G_Last_Denial_Code := 2;
        GVL_ALARM_AUDIBLE_ACK.G_Status_Text := 'Audible acknowledgement denied: access level < 2';
    ELSIF GVL_ALARM_AUDIBLE_ACK.G_Ack_Count_Current_Alarm >= 3 THEN
        GVL_ALARM_AUDIBLE_ACK.G_Last_Ack_Denied := TRUE;
        GVL_ALARM_AUDIBLE_ACK.G_Last_Denial_Code := 3;
        GVL_ALARM_AUDIBLE_ACK.G_Ack_Limit_Reached := TRUE;
        GVL_ALARM_AUDIBLE_ACK.G_Status_Text := 'Audible acknowledgement denied: limit reached';
    ELSE
        GVL_ALARM_AUDIBLE_ACK.G_Ack_Count_Current_Alarm := GVL_ALARM_AUDIBLE_ACK.G_Ack_Count_Current_Alarm + 1;
        GVL_ALARM_AUDIBLE_ACK.G_Ack_Active := TRUE;
        GVL_ALARM_AUDIBLE_ACK.G_Ack_Expires_MS := GVL_TIME_SERVICE.G_Now_MS + (GVL_CONSTANTS.C_MS_IN_MINUTE * 5);
        GVL_ALARM_AUDIBLE_ACK.G_Ack_Remaining_MS := GVL_CONSTANTS.C_MS_IN_MINUTE * 5;
        GVL_ALARM_AUDIBLE_ACK.G_Last_Ack_Accepted := TRUE;
        GVL_ALARM_AUDIBLE_ACK.G_Last_Event_MS := GVL_TIME_SERVICE.G_Now_MS;
        GVL_ALARM_AUDIBLE_ACK.G_Status_Text := 'Audible alarm acknowledged for 5 minutes';
    END_IF;

    GVL_ALARM_AUDIBLE_ACK.G_Ack_Request := FALSE;
END_IF;

IF GVL_ALARM_AUDIBLE_ACK.G_Ack_Count_Current_Alarm >= 3 THEN
    GVL_ALARM_AUDIBLE_ACK.G_Ack_Limit_Reached := TRUE;
ELSE
    GVL_ALARM_AUDIBLE_ACK.G_Ack_Limit_Reached := FALSE;
END_IF;

// >>> BULK_SYNC_ANCHOR: PRG_Alarm_Audible_Ack_Manager <<<
END_PROGRAM

(* ---- PRG_Authority_Lineage_Governor.st ---- *)
PROGRAM PRG_Authority_Lineage_Governor
VAR
    L_Now_MS : UDINT;
    L_Lineage_Valid : BOOL := TRUE;
    L_Error_Code : UDINT := 0;
    L_Error_Text : STRING(160) := '';
END_VAR

L_Now_MS := GVL_STATUS.G_System_Time_MS;
L_Lineage_Valid := TRUE;
L_Error_Code := 0;
L_Error_Text := '';

// Fail-safe defaults.
GVL_AUTHORITY_LINEAGE.Authority_Lineage_Valid := FALSE;
GVL_AUTHORITY_LINEAGE.Warm_Restart_Continuity_Valid := FALSE;
GVL_AUTHORITY_LINEAGE.HA_Resume_Continuity_Valid := FALSE;
GVL_AUTHORITY_LINEAGE.Retained_State_Integrity_Valid := FALSE;

// Replay detection.
IF GVL_AUTHORITY_LINEAGE.Authority_Replay_Suspected THEN
    L_Lineage_Valid := FALSE;
    L_Error_Code := 25000;
    L_Error_Text := 'Authority replay suspected';
END_IF;

IF L_Lineage_Valid
AND GVL_AUTHORITY_LINEAGE.Retained_State_Skew_Detected THEN
    L_Lineage_Valid := FALSE;
    L_Error_Code := 25001;
    L_Error_Text := 'Retained state skew detected';
END_IF;

IF L_Lineage_Valid
AND GVL_AUTHORITY_LINEAGE.Partial_Authority_Resurrection_Detected THEN
    L_Lineage_Valid := FALSE;
    L_Error_Code := 25002;
    L_Error_Text := 'Partial authority resurrection detected';
END_IF;

IF L_Lineage_Valid
AND GVL_AUTHORITY_LINEAGE.Epoch_Lineage_Discontinuity_Detected THEN
    L_Lineage_Valid := FALSE;
    L_Error_Code := 25003;
    L_Error_Text := 'Epoch lineage discontinuity detected';
END_IF;

// Physical authority epoch continuity.
IF L_Lineage_Valid
AND (GVL_PHYSICAL_AUTHORITY_EPOCH.Physical_Authority_Epoch <
     GVL_AUTHORITY_LINEAGE.Last_Physical_Authority_Epoch) THEN

    GVL_AUTHORITY_LINEAGE.Authority_Replay_Suspected := TRUE;

    L_Lineage_Valid := FALSE;
    L_Error_Code := 25010;
    L_Error_Text := 'Physical authority epoch rollback detected';
END_IF;

// Runtime epoch continuity.
IF L_Lineage_Valid
AND (GVL_RUNTIME_EPOCH.Runtime_Epoch <
     GVL_AUTHORITY_LINEAGE.Last_Runtime_Epoch) THEN

    GVL_AUTHORITY_LINEAGE.Retained_State_Skew_Detected := TRUE;

    L_Lineage_Valid := FALSE;
    L_Error_Code := 25011;
    L_Error_Text := 'Runtime epoch rollback detected';
END_IF;

// Output publication continuity.
IF L_Lineage_Valid
AND (GVL_OUTPUT_EPOCH.Output_Publication_Epoch <
     GVL_AUTHORITY_LINEAGE.Last_Output_Publication_Epoch) THEN

    GVL_AUTHORITY_LINEAGE.Partial_Authority_Resurrection_Detected := TRUE;

    L_Lineage_Valid := FALSE;
    L_Error_Code := 25012;
    L_Error_Text := 'Output publication epoch rollback detected';
END_IF;

IF L_Lineage_Valid THEN
    GVL_AUTHORITY_LINEAGE.Authority_Lineage_Valid := TRUE;

    GVL_AUTHORITY_LINEAGE.Warm_Restart_Continuity_Valid := TRUE;
    GVL_AUTHORITY_LINEAGE.HA_Resume_Continuity_Valid := TRUE;
    GVL_AUTHORITY_LINEAGE.Retained_State_Integrity_Valid := TRUE;

    GVL_AUTHORITY_LINEAGE.Authority_Lineage_Epoch :=
        GVL_PHYSICAL_AUTHORITY_EPOCH.Physical_Authority_Epoch;

    GVL_AUTHORITY_LINEAGE.Last_Physical_Authority_Epoch :=
        GVL_PHYSICAL_AUTHORITY_EPOCH.Physical_Authority_Epoch;

    GVL_AUTHORITY_LINEAGE.Last_Runtime_Epoch :=
        GVL_RUNTIME_EPOCH.Runtime_Epoch;

    GVL_AUTHORITY_LINEAGE.Last_Output_Publication_Epoch :=
        GVL_OUTPUT_EPOCH.Output_Publication_Epoch;

    GVL_AUTHORITY_LINEAGE.Authority_Lineage_Last_Update_MS := L_Now_MS;

    GVL_AUTHORITY_LINEAGE.Authority_Lineage_Last_Error_Code := 0;
    GVL_AUTHORITY_LINEAGE.Authority_Lineage_Last_Error_Text := '';
ELSE
    GVL_AUTHORITY_LINEAGE.Authority_Lineage_Valid := FALSE;

    GVL_AUTHORITY_LINEAGE.Authority_Lineage_Last_Error_Code := L_Error_Code;
    GVL_AUTHORITY_LINEAGE.Authority_Lineage_Last_Error_Text := L_Error_Text;

    GVL_AUTHORITY_LINEAGE.Authority_Lineage_Invalidation_Count :=
        GVL_AUTHORITY_LINEAGE.Authority_Lineage_Invalidation_Count + 1;
END_IF;

END_PROGRAM

(* ---- PRG_Authority_Resurrection_Boundary_Governor.st ---- *)
PROGRAM PRG_Authority_Resurrection_Boundary_Governor
IF GVL_RECOVERY_REACTIVATION_CONTROL_FABRIC.Recovery_Reactivation_Control_Granted
AND NOT GVL_AUTHORITY_RESURRECTION_BOUNDARY_FABRIC.Partial_Recovery_Authority_Leak
AND NOT GVL_AUTHORITY_RESURRECTION_BOUNDARY_FABRIC.Unsafe_Authority_Resurrection_Detected
AND NOT GVL_AUTHORITY_RESURRECTION_BOUNDARY_FABRIC.Resurrection_Authority_Fork_Detected THEN

    GVL_AUTHORITY_RESURRECTION_BOUNDARY_FABRIC.Authority_Resurrection_Boundary_Valid := TRUE;
    GVL_AUTHORITY_RESURRECTION_BOUNDARY_FABRIC.Authority_Resurrection_Bounded := TRUE;
    GVL_AUTHORITY_RESURRECTION_BOUNDARY_FABRIC.Authority_Recovery_Lineage_Stable := TRUE;
    GVL_AUTHORITY_RESURRECTION_BOUNDARY_FABRIC.Distributed_Authority_Recovery_Consensus := TRUE;
END_IF;
END_PROGRAM

(* ---- PRG_Authority_Revocation_Governor.st ---- *)
PROGRAM PRG_Authority_Revocation_Governor
VAR
    L_Now_MS : UDINT;
    L_Revocation_Required : BOOL := FALSE;
END_VAR

L_Now_MS := GVL_STATUS.G_System_Time_MS;

// Fail-safe defaults.
GVL_AUTHORITY_REVOCATION.Authority_Revocation_Active := FALSE;
GVL_AUTHORITY_REVOCATION.Authority_Revocation_Propagated := FALSE;
GVL_AUTHORITY_REVOCATION.Authority_Fail_Closed_Valid := FALSE;
GVL_AUTHORITY_REVOCATION.Revocation_Order_Valid := FALSE;

// Detect upstream authority invalidation.
GVL_AUTHORITY_REVOCATION.Snapshot_Authority_Revoked :=
    NOT GVL_PHYSICAL_SNAPSHOT.Physical_Snapshot_Valid;

GVL_AUTHORITY_REVOCATION.Sensor_Consensus_Authority_Revoked :=
    NOT GVL_SENSOR_CONSENSUS.Sensor_Consensus_Valid;

GVL_AUTHORITY_REVOCATION.Telemetry_Causality_Authority_Revoked :=
    NOT GVL_TELEMETRY.Command_Telemetry_Causality_Valid;

GVL_AUTHORITY_REVOCATION.Physical_Authority_Epoch_Revoked :=
    NOT GVL_PHYSICAL_AUTHORITY_EPOCH.Physical_Authority_Epoch_Valid;

GVL_AUTHORITY_REVOCATION.Authority_Lineage_Revoked :=
    NOT GVL_AUTHORITY_LINEAGE.Authority_Lineage_Valid;

L_Revocation_Required :=
    GVL_AUTHORITY_REVOCATION.Snapshot_Authority_Revoked
    OR GVL_AUTHORITY_REVOCATION.Sensor_Consensus_Authority_Revoked
    OR GVL_AUTHORITY_REVOCATION.Telemetry_Causality_Authority_Revoked
    OR GVL_AUTHORITY_REVOCATION.Physical_Authority_Epoch_Revoked
    OR GVL_AUTHORITY_REVOCATION.Authority_Lineage_Revoked;

IF L_Revocation_Required THEN
    GVL_AUTHORITY_REVOCATION.Authority_Revocation_Active := TRUE;
    GVL_AUTHORITY_REVOCATION.Quarantine_Fabric_Active := TRUE;

    GVL_AUTHORITY_REVOCATION.PreOutput_Authority_Revoked := TRUE;
    GVL_AUTHORITY_REVOCATION.Physical_IO_Release_Denied := TRUE;

    GVL_AUTHORITY_REVOCATION.Authority_Revocation_Propagated := TRUE;
    GVL_AUTHORITY_REVOCATION.Authority_Fail_Closed_Valid := TRUE;
    GVL_AUTHORITY_REVOCATION.Revocation_Order_Valid := TRUE;

    GVL_AUTHORITY_REVOCATION.Revocation_Epoch :=
        GVL_PHYSICAL_AUTHORITY_EPOCH.Physical_Authority_Epoch;

    GVL_AUTHORITY_REVOCATION.Revocation_Last_Update_MS := L_Now_MS;
ELSE
    GVL_AUTHORITY_REVOCATION.Authority_Revocation_Active := FALSE;
    GVL_AUTHORITY_REVOCATION.Quarantine_Fabric_Active := FALSE;

    GVL_AUTHORITY_REVOCATION.PreOutput_Authority_Revoked := FALSE;
    GVL_AUTHORITY_REVOCATION.Physical_IO_Release_Denied := FALSE;

    GVL_AUTHORITY_REVOCATION.Authority_Revocation_Propagated := FALSE;
    GVL_AUTHORITY_REVOCATION.Authority_Fail_Closed_Valid := TRUE;
    GVL_AUTHORITY_REVOCATION.Revocation_Order_Valid := TRUE;
END_IF;

END_PROGRAM

(* ---- PRG_Away_Heating_HMI_Applicator.st ---- *)
PROGRAM PRG_Away_Heating_HMI_Applicator
VAR
    L_Circuit : INT;
    L_Delay_MS : UDINT;
    L_Preheat_Lead_MS : UDINT;
    L_Return_Grace_MS : UDINT;
END_VAR

// HMI per-circuit profile update.
IF GVL_AWAY_HEATING_HMI.G_Set_Circuit_Profile_Req THEN
    L_Circuit := GVL_AWAY_HEATING_HMI.G_Profile_Circuit;

    IF (L_Circuit >= 1) AND (L_Circuit <= GVL_CONSTANTS.C_MAX_HEATING_CIRCUITS) THEN
        IF (GVL_AWAY_HEATING_HMI.G_Profile_Comfort_Temp >= REAL#5.0) AND
           (GVL_AWAY_HEATING_HMI.G_Profile_Comfort_Temp <= REAL#30.0) AND
           (GVL_AWAY_HEATING_HMI.G_Profile_Economy_Temp >= REAL#5.0) AND
           (GVL_AWAY_HEATING_HMI.G_Profile_Economy_Temp <= GVL_AWAY_HEATING_HMI.G_Profile_Comfort_Temp) AND
           (GVL_AWAY_HEATING_HMI.G_Profile_Long_Away_Temp >= REAL#5.0) AND
           (GVL_AWAY_HEATING_HMI.G_Profile_Long_Away_Temp <= GVL_AWAY_HEATING_HMI.G_Profile_Economy_Temp) THEN

            GVL_CONFIG.G_HMI_FloorHeating_Configs[L_Circuit].use_in_normal := GVL_AWAY_HEATING_HMI.G_Profile_Use_In_Normal;
            GVL_CONFIG.G_HMI_FloorHeating_Configs[L_Circuit].use_in_away_preheat := GVL_AWAY_HEATING_HMI.G_Profile_Use_In_Away_Preheat;
            GVL_CONFIG.G_HMI_FloorHeating_Configs[L_Circuit].comfort_temp := GVL_AWAY_HEATING_HMI.G_Profile_Comfort_Temp;
            GVL_CONFIG.G_HMI_FloorHeating_Configs[L_Circuit].economy_temp := GVL_AWAY_HEATING_HMI.G_Profile_Economy_Temp;
            GVL_CONFIG.G_HMI_FloorHeating_Configs[L_Circuit].long_away_temp := GVL_AWAY_HEATING_HMI.G_Profile_Long_Away_Temp;
            GVL_CONFIG.G_HMI_FloorHeating_Configs[L_Circuit].design_temp := GVL_AWAY_HEATING_HMI.G_Profile_Comfort_Temp;

            GVL_AWAY_HEATING_HMI.G_Last_Error := FALSE;
            GVL_AWAY_HEATING_HMI.G_Last_Status_Text := 'Away heating profile applied';
        ELSE
            GVL_AWAY_HEATING_HMI.G_Last_Error := TRUE;
            GVL_AWAY_HEATING_HMI.G_Last_Status_Text := 'Away heating profile rejected: invalid temperatures';
        END_IF;
    ELSE
        GVL_AWAY_HEATING_HMI.G_Last_Error := TRUE;
        GVL_AWAY_HEATING_HMI.G_Last_Status_Text := 'Away heating profile rejected: invalid circuit';
    END_IF;

    GVL_AWAY_HEATING_HMI.G_Last_Update_MS := GVL_TIME_SERVICE.G_Now_MS;
    GVL_AWAY_HEATING_HMI.G_Set_Circuit_Profile_Req := FALSE;
END_IF;

// Gateway compatibility: CMD_SET_TEMP updates comfort temperature for one circuit.
IF GVL_INTENT_USER.I_Set_Temp_Req THEN
    L_Circuit := GVL_INTENT_USER.I_Target_Zone;

    IF (L_Circuit >= 1) AND (L_Circuit <= GVL_CONSTANTS.C_MAX_HEATING_CIRCUITS) AND
       (GVL_INTENT_USER.I_Target_Temperature >= REAL#5.0) AND
       (GVL_INTENT_USER.I_Target_Temperature <= REAL#30.0) THEN
        GVL_CONFIG.G_HMI_FloorHeating_Configs[L_Circuit].comfort_temp := GVL_INTENT_USER.I_Target_Temperature;
        GVL_CONFIG.G_HMI_FloorHeating_Configs[L_Circuit].design_temp := GVL_INTENT_USER.I_Target_Temperature;

        IF GVL_CONFIG.G_HMI_FloorHeating_Configs[L_Circuit].economy_temp <= REAL#0.0 THEN
            GVL_CONFIG.G_HMI_FloorHeating_Configs[L_Circuit].economy_temp := GVL_INTENT_USER.I_Target_Temperature - REAL#3.0;
        END_IF;

        IF GVL_CONFIG.G_HMI_FloorHeating_Configs[L_Circuit].long_away_temp <= REAL#0.0 THEN
            GVL_CONFIG.G_HMI_FloorHeating_Configs[L_Circuit].long_away_temp := GVL_POLICY.G_Away_Long_Economy_Setpoint_C;
        END_IF;
    END_IF;
END_IF;

// HMI planned return update. Delay is relative to current monotonic PLC time.
IF GVL_AWAY_HEATING_HMI.G_Set_Planned_Return_Req THEN
    IF GVL_AWAY_HEATING_HMI.G_Planned_Return_Enabled AND (GVL_AWAY_HEATING_HMI.G_Planned_Return_Delay_Hours > REAL#0.0) THEN
        L_Delay_MS := REAL_TO_UDINT(GVL_AWAY_HEATING_HMI.G_Planned_Return_Delay_Hours * REAL#3600000.0);
        L_Preheat_Lead_MS := REAL_TO_UDINT(GVL_AWAY_HEATING_HMI.G_Preheat_Lead_Hours * REAL#3600000.0);
        L_Return_Grace_MS := REAL_TO_UDINT(GVL_AWAY_HEATING_HMI.G_Return_Grace_Hours * REAL#3600000.0);

        IF L_Preheat_Lead_MS = 0 THEN
            L_Preheat_Lead_MS := 10800000;
        END_IF;
        IF L_Return_Grace_MS = 0 THEN
            L_Return_Grace_MS := 86400000;
        END_IF;

        GVL_POLICY.G_Away_Planned_Return_Enabled := TRUE;
        GVL_POLICY.G_Away_Planned_Return_MS := GVL_TIME_SERVICE.G_Now_MS + L_Delay_MS;
        GVL_POLICY.G_Away_Preheat_Lead_MS := L_Preheat_Lead_MS;
        GVL_POLICY.G_Away_Return_Grace_MS := L_Return_Grace_MS;
        GVL_POLICY.G_Away_Return_Expired := FALSE;
        GVL_POLICY.G_Away_Return_Grace_Active := FALSE;
        GVL_POLICY.G_Away_Return_Preheat_Active := FALSE;

        GVL_AWAY_HEATING_HMI.G_Last_Error := FALSE;
        GVL_AWAY_HEATING_HMI.G_Last_Status_Text := 'Planned return configured';
    ELSE
        GVL_POLICY.G_Away_Planned_Return_Enabled := FALSE;
        GVL_POLICY.G_Away_Return_Preheat_Active := FALSE;
        GVL_POLICY.G_Away_Return_Grace_Active := FALSE;
        GVL_POLICY.G_Away_Return_Expired := FALSE;

        GVL_AWAY_HEATING_HMI.G_Last_Error := FALSE;
        GVL_AWAY_HEATING_HMI.G_Last_Status_Text := 'Planned return disabled';
    END_IF;

    GVL_AWAY_HEATING_HMI.G_Last_Update_MS := GVL_TIME_SERVICE.G_Now_MS;
    GVL_AWAY_HEATING_HMI.G_Set_Planned_Return_Req := FALSE;
END_IF;

IF GVL_AWAY_HEATING_HMI.G_Clear_Planned_Return_Req THEN
    GVL_POLICY.G_Away_Planned_Return_Enabled := FALSE;
    GVL_POLICY.G_Away_Return_Preheat_Active := FALSE;
    GVL_POLICY.G_Away_Return_Grace_Active := FALSE;
    GVL_POLICY.G_Away_Return_Expired := FALSE;
    GVL_AWAY_HEATING_HMI.G_Last_Error := FALSE;
    GVL_AWAY_HEATING_HMI.G_Last_Status_Text := 'Planned return cleared';
    GVL_AWAY_HEATING_HMI.G_Last_Update_MS := GVL_TIME_SERVICE.G_Now_MS;
    GVL_AWAY_HEATING_HMI.G_Clear_Planned_Return_Req := FALSE;
END_IF;

// Gateway compatibility: CMD_SET_CONFIG with target_zone=0 configures/clears planned return.
IF GVL_INTENT_USER.I_Set_Config_Req AND
   (GVL_GATEWAY.G_Gateway_Command.command_type = E_Gateway_Command_Type.CMD_SET_CONFIG) AND
   (GVL_GATEWAY.G_Gateway_Command.target_zone = 0) THEN
    IF GVL_GATEWAY.G_Gateway_Command.target_on_off AND (GVL_GATEWAY.G_Gateway_Command.target_value > REAL#0.0) THEN
        L_Delay_MS := REAL_TO_UDINT(GVL_GATEWAY.G_Gateway_Command.target_value * REAL#3600000.0);
        GVL_POLICY.G_Away_Planned_Return_Enabled := TRUE;
        GVL_POLICY.G_Away_Planned_Return_MS := GVL_TIME_SERVICE.G_Now_MS + L_Delay_MS;
        GVL_POLICY.G_Away_Return_Expired := FALSE;
        GVL_POLICY.G_Away_Return_Grace_Active := FALSE;
        GVL_POLICY.G_Away_Return_Preheat_Active := FALSE;
    ELSE
        GVL_POLICY.G_Away_Planned_Return_Enabled := FALSE;
        GVL_POLICY.G_Away_Return_Preheat_Active := FALSE;
        GVL_POLICY.G_Away_Return_Grace_Active := FALSE;
        GVL_POLICY.G_Away_Return_Expired := FALSE;
    END_IF;
END_IF;

END_PROGRAM

(* ---- PRG_Away_Restore_Manager.st ---- *)
PROGRAM PRG_Away_Restore_Manager
VAR
    L_i : INT;
    L_Away_Active_Prev : BOOL := FALSE;
    L_Away_Level_Prev : BYTE := 0;
    L_Take_Snapshot : BOOL;
    L_Start_Restore : BOOL;
END_VAR

L_Take_Snapshot :=
    GVL_POLICY.G_Away_Active AND
    (GVL_POLICY.G_Away_Level = 1) AND
    (NOT L_Away_Active_Prev);

IF L_Take_Snapshot THEN
    FOR L_i := 1 TO GVL_CONSTANTS.C_MAX_LIGHT_ZONES DO
        GVL_AWAY_RESTORE.G_Lighting_Levels[L_i] := GVL_STATE.G_Lighting_Levels[L_i];
    END_FOR;

    FOR L_i := 1 TO GVL_CONSTANTS.C_MAX_SOCKETS DO
        GVL_AWAY_RESTORE.G_Socket_States[L_i] := GVL_STATE.G_Socket_States[L_i];
    END_FOR;

    GVL_AWAY_RESTORE.G_Snapshot_Valid := TRUE;
    GVL_AWAY_RESTORE.G_Snapshot_Taken_MS := GVL_TIME_SERVICE.G_Now_MS;
    GVL_AWAY_RESTORE.G_Restore_Done := FALSE;
END_IF;

L_Start_Restore :=
    GVL_POLICY.G_Away_Restore_Requested AND
    GVL_AWAY_RESTORE.G_Snapshot_Valid;

IF L_Start_Restore THEN
    GVL_AWAY_RESTORE.G_Restore_Active := TRUE;
    GVL_AWAY_RESTORE.G_Restore_Started_MS := GVL_TIME_SERVICE.G_Now_MS;
    GVL_AWAY_RESTORE.G_Restore_Done := FALSE;
END_IF;

IF GVL_AWAY_RESTORE.G_Restore_Active THEN
    GVL_AWAY_RESTORE.G_Restore_Progress := GVL_POLICY.G_Away_Restore_Progress;

    IF NOT GVL_POLICY.G_Away_Restore_Active THEN
        GVL_AWAY_RESTORE.G_Restore_Progress := 1.0;
        GVL_AWAY_RESTORE.G_Restore_Active := FALSE;
        GVL_AWAY_RESTORE.G_Restore_Done := TRUE;
        GVL_AWAY_RESTORE.G_Snapshot_Valid := FALSE;
    END_IF;
ELSE
    IF NOT GVL_AWAY_RESTORE.G_Restore_Done THEN
        GVL_AWAY_RESTORE.G_Restore_Progress := 0.0;
    END_IF;
END_IF;

L_Away_Active_Prev := GVL_POLICY.G_Away_Active;
L_Away_Level_Prev := GVL_POLICY.G_Away_Level;

END_PROGRAM

(* ---- PRG_Behavior_Adapt_Profile.st ---- *)
PROGRAM PRG_Behavior_Adapt_Profile

// Centralized tuning profile controller.
// This block enforces consistent adaptive behavior settings.

CASE GVL_BEHAVIOR_ADAPT.G_Adapt_Profile OF

    ADAPT_PROFILE_STABLE:
        GVL_BEHAVIOR_ADAPT.G_Adapt_Learning_Rate := 0.03;
        GVL_BEHAVIOR_ADAPT.G_Confidence_Learning_Rate := 0.03;
        GVL_BEHAVIOR_ADAPT.G_Decay_Factor := 0.998;
        GVL_BEHAVIOR_ADAPT.G_Adapt_Update_Threshold := 7;

    ADAPT_PROFILE_BALANCED:
        GVL_BEHAVIOR_ADAPT.G_Adapt_Learning_Rate := 0.05;
        GVL_BEHAVIOR_ADAPT.G_Confidence_Learning_Rate := 0.05;
        GVL_BEHAVIOR_ADAPT.G_Decay_Factor := 0.995;
        GVL_BEHAVIOR_ADAPT.G_Adapt_Update_Threshold := 5;

    ADAPT_PROFILE_AGGRESSIVE:
        GVL_BEHAVIOR_ADAPT.G_Adapt_Learning_Rate := 0.08;
        GVL_BEHAVIOR_ADAPT.G_Confidence_Learning_Rate := 0.08;
        GVL_BEHAVIOR_ADAPT.G_Decay_Factor := 0.990;
        GVL_BEHAVIOR_ADAPT.G_Adapt_Update_Threshold := 3;

END_CASE;

// >>> BULK_SYNC_ANCHOR: PRG_Behavior_Adapt_Profile <<<

(* ---- PRG_Command_Arbitration.st ---- *)
PROGRAM PRG_Command_Arbitration
// ==============================================================================
// COMMAND ARBITRATION — deterministic command-shadow phase map.
// ==============================================================================
// Execution preserves the former priority model:
// 1. reset + PLC role guard
// 2. safety mode projection
// 3. safe user/rule projection and conflict cleanup
// 4. single deterministic write into GVL_COMMAND_SHADOW
// ==============================================================================

PRG_Command_Arbitration_Phase_01_Reset_Role();

IF GVL_COMMAND_ARBITRATION_BUFFER.B_Role_Conflict_Active
   OR GVL_COMMAND_ARBITRATION_BUFFER.B_PLC_Inactive_Active THEN
    PRG_Command_Arbitration_Phase_04_Write_Shadow();
    RETURN;
END_IF;

PRG_Command_Arbitration_Phase_02_Safety_Mode();
PRG_Command_Arbitration_Phase_03_User_Rules_Conflict();
PRG_Command_Arbitration_Phase_04_Write_Shadow();

// >>> BULK_SYNC_ANCHOR: PRG_Command_Arbitration <<<
END_PROGRAM

(* ---- PRG_Command_Arbitration_Phase_02_Safety_Mode.st ---- *)
PROGRAM PRG_Command_Arbitration_Phase_02_Safety_Mode
// Command arbitration phase 02: project safety mode into deterministic buffer.

GVL_COMMAND_ARBITRATION_BUFFER.B_Mode := GVL_SAFETY_SHUTDOWN.G_Safety_Mode;
GVL_COMMAND_ARBITRATION_BUFFER.B_Safety_Active := FALSE;

CASE GVL_COMMAND_ARBITRATION_BUFFER.B_Mode OF

    NORMAL:
        GVL_COMMAND_ARBITRATION_BUFFER.B_Safety_Active := FALSE;

    FIRE:
        GVL_COMMAND_ARBITRATION_BUFFER.B_Safety_Active := TRUE;
        GVL_COMMAND_ARBITRATION_BUFFER.B_Heating_Block := GVL_COMMAND_POLICY_CONFIG.G_Fire_Block_Heating;
        GVL_COMMAND_ARBITRATION_BUFFER.B_Boiler_Stop := GVL_COMMAND_POLICY_CONFIG.G_Fire_Stop_Boiler;
        GVL_COMMAND_ARBITRATION_BUFFER.B_Vent_Stop := FALSE;
        GVL_COMMAND_ARBITRATION_BUFFER.B_Vent_PV3_Boost := FALSE;
        GVL_COMMAND_ARBITRATION_BUFFER.B_Exhaust_100_Req := FALSE;
        GVL_COMMAND_ARBITRATION_BUFFER.B_Vent_Smoke_Exhaust := TRUE;
        GVL_COMMAND_ARBITRATION_BUFFER.B_Heating_Emergency_Stop := GVL_COMMAND_POLICY_CONFIG.G_Fire_Block_Heating;
        GVL_COMMAND_ARBITRATION_BUFFER.B_Lock_1_Open := GVL_COMMAND_POLICY_CONFIG.G_Fire_Open_Lock_1;
        GVL_COMMAND_ARBITRATION_BUFFER.B_Lock_2_Open := GVL_COMMAND_POLICY_CONFIG.G_Fire_Open_Lock_2;
        GVL_COMMAND_ARBITRATION_BUFFER.B_Gate_Open := GVL_COMMAND_POLICY_CONFIG.G_Fire_Open_Gate;
        GVL_COMMAND_ARBITRATION_BUFFER.B_Wicket_Open := GVL_COMMAND_POLICY_CONFIG.G_Fire_Open_Wicket;

    GAS:
        GVL_COMMAND_ARBITRATION_BUFFER.B_Safety_Active := TRUE;
        GVL_COMMAND_ARBITRATION_BUFFER.B_Gas_Valve_Close := GVL_COMMAND_POLICY_CONFIG.G_Gas_Close_Gas;
        GVL_COMMAND_ARBITRATION_BUFFER.B_Boiler_Stop := GVL_COMMAND_POLICY_CONFIG.G_Gas_Stop_Boiler;
        GVL_COMMAND_ARBITRATION_BUFFER.B_Heating_Block := GVL_COMMAND_POLICY_CONFIG.G_Gas_Block_Heating;
        GVL_COMMAND_ARBITRATION_BUFFER.B_Heating_Gas_Safety_Stop := GVL_COMMAND_POLICY_CONFIG.G_Gas_Block_Heating;
        GVL_COMMAND_ARBITRATION_BUFFER.B_Vent_PV3_Boost := TRUE;
        GVL_COMMAND_ARBITRATION_BUFFER.B_Vent_Smoke_Exhaust := FALSE;
        GVL_COMMAND_ARBITRATION_BUFFER.B_Gate_Open := GVL_COMMAND_POLICY_CONFIG.G_Gas_Open_Gate;
        GVL_COMMAND_ARBITRATION_BUFFER.B_Wicket_Open := GVL_COMMAND_POLICY_CONFIG.G_Gas_Open_Wicket;
        GVL_COMMAND_ARBITRATION_BUFFER.B_Lock_1_Open := GVL_COMMAND_POLICY_CONFIG.G_Gas_Open_Lock_1;
        GVL_COMMAND_ARBITRATION_BUFFER.B_Lock_2_Open := GVL_COMMAND_POLICY_CONFIG.G_Gas_Open_Lock_2;

    WATER_LEAK:
        GVL_COMMAND_ARBITRATION_BUFFER.B_Safety_Active := TRUE;
        GVL_COMMAND_ARBITRATION_BUFFER.B_Water_Block := GVL_COMMAND_POLICY_CONFIG.G_Water_Block_Water;
        GVL_COMMAND_ARBITRATION_BUFFER.B_Water_Emergency_Stop := GVL_COMMAND_POLICY_CONFIG.G_Water_Block_Water;
        GVL_COMMAND_ARBITRATION_BUFFER.B_Close_Valve_35 := GVL_COMMAND_POLICY_CONFIG.G_Water_Block_Water;
        GVL_COMMAND_ARBITRATION_BUFFER.B_Close_Valve_36 := GVL_COMMAND_POLICY_CONFIG.G_Water_Block_Water;

    GLOBAL_STOP:
        GVL_COMMAND_ARBITRATION_BUFFER.B_Safety_Active := TRUE;
        GVL_COMMAND_ARBITRATION_BUFFER.B_Heating_Block := GVL_COMMAND_POLICY_CONFIG.G_GlobalStop_Block_Heating;
        GVL_COMMAND_ARBITRATION_BUFFER.B_Heating_Emergency_Stop := GVL_COMMAND_POLICY_CONFIG.G_GlobalStop_Block_Heating;
        GVL_COMMAND_ARBITRATION_BUFFER.B_Boiler_Stop := GVL_COMMAND_POLICY_CONFIG.G_GlobalStop_Stop_Boiler;
        GVL_COMMAND_ARBITRATION_BUFFER.B_Vent_Stop := GVL_COMMAND_POLICY_CONFIG.G_GlobalStop_Stop_Vent;
        GVL_COMMAND_ARBITRATION_BUFFER.B_Water_Block := GVL_COMMAND_POLICY_CONFIG.G_GlobalStop_Block_Water;
        GVL_COMMAND_ARBITRATION_BUFFER.B_Water_Emergency_Stop := GVL_COMMAND_POLICY_CONFIG.G_GlobalStop_Block_Water;
        GVL_COMMAND_ARBITRATION_BUFFER.B_Close_Valve_35 := GVL_COMMAND_POLICY_CONFIG.G_GlobalStop_Block_Water;
        GVL_COMMAND_ARBITRATION_BUFFER.B_Close_Valve_36 := GVL_COMMAND_POLICY_CONFIG.G_GlobalStop_Block_Water;

ELSE
        GVL_COMMAND_ARBITRATION_BUFFER.B_Safety_Active := TRUE;
        GVL_COMMAND_ARBITRATION_BUFFER.B_Gas_Valve_Close := TRUE;
        GVL_COMMAND_ARBITRATION_BUFFER.B_Boiler_Stop := TRUE;
        GVL_COMMAND_ARBITRATION_BUFFER.B_Heating_Block := TRUE;
        GVL_COMMAND_ARBITRATION_BUFFER.B_Heating_Emergency_Stop := TRUE;
        GVL_COMMAND_ARBITRATION_BUFFER.B_Vent_Stop := TRUE;
        GVL_COMMAND_ARBITRATION_BUFFER.B_Water_Block := TRUE;
        GVL_COMMAND_ARBITRATION_BUFFER.B_Water_Emergency_Stop := TRUE;
        GVL_COMMAND_ARBITRATION_BUFFER.B_Close_Valve_35 := TRUE;
        GVL_COMMAND_ARBITRATION_BUFFER.B_Close_Valve_36 := TRUE;
END_CASE;

// >>> BULK_SYNC_ANCHOR: PRG_Command_Arbitration_Phase_02_Safety_Mode <<<
END_PROGRAM

(* ---- PRG_Command_Arbitration_Phase_03_User_Rules_Conflict.st ---- *)
PROGRAM PRG_Command_Arbitration_Phase_03_User_Rules_Conflict
// Command arbitration phase 03: user intent, automation rules and conflict cleanup.
VAR
    L_i : INT;
END_VAR

GVL_COMMAND_ARBITRATION_BUFFER.B_User_Access_OK :=
    GVL_INTENT_USER.I_Source_Valid
    AND (GVL_INTENT_USER.I_User_Access_Level >= 2);

IF (NOT GVL_COMMAND_ARBITRATION_BUFFER.B_Safety_Active)
   AND GVL_COMMAND_ARBITRATION_BUFFER.B_User_Access_OK THEN

    IF GVL_INTENT_USER.I_Lock_1_Open_Request THEN
        GVL_COMMAND_ARBITRATION_BUFFER.B_Lock_1_Open := TRUE;
        GVL_COMMAND_ARBITRATION_BUFFER.B_Lock_1_Close := FALSE;
    ELSIF GVL_INTENT_USER.I_Lock_1_Close_Request THEN
        GVL_COMMAND_ARBITRATION_BUFFER.B_Lock_1_Open := FALSE;
        GVL_COMMAND_ARBITRATION_BUFFER.B_Lock_1_Close := TRUE;
    END_IF;

    IF GVL_INTENT_USER.I_Lock_2_Open_Request THEN
        GVL_COMMAND_ARBITRATION_BUFFER.B_Lock_2_Open := TRUE;
        GVL_COMMAND_ARBITRATION_BUFFER.B_Lock_2_Close := FALSE;
    ELSIF GVL_INTENT_USER.I_Lock_2_Close_Request THEN
        GVL_COMMAND_ARBITRATION_BUFFER.B_Lock_2_Open := FALSE;
        GVL_COMMAND_ARBITRATION_BUFFER.B_Lock_2_Close := TRUE;
    END_IF;

    IF GVL_INTENT_USER.I_Gate_Open_Request THEN
        GVL_COMMAND_ARBITRATION_BUFFER.B_Gate_Open := TRUE;
    END_IF;

    IF GVL_INTENT_USER.I_Wicket_Open_Request THEN
        GVL_COMMAND_ARBITRATION_BUFFER.B_Wicket_Open := TRUE;
    END_IF;
END_IF;

// Dangerous user actions require explicit confirmation and elevated access.
IF (NOT GVL_COMMAND_ARBITRATION_BUFFER.B_Safety_Active)
   AND GVL_INTENT_USER.I_Source_Valid
   AND GVL_INTENT_USER.I_Dangerous_Action_Request
   AND GVL_INTENT_USER.I_Dangerous_Action_Confirm
   AND (GVL_INTENT_USER.I_User_Access_Level >= 2) THEN
    // Reserved for future high-risk manual actions.
    // No direct safety override is allowed here.
END_IF;

IF NOT GVL_COMMAND_ARBITRATION_BUFFER.B_Safety_Active THEN
    FOR L_i := 1 TO GVL_CONSTANTS.C_MAX_RULES DO
        IF GVL_STATE.G_Rule_Actions[L_i].Active AND GVL_STATE.G_Rule_Actions[L_i].Triggered THEN
            CASE GVL_STATE.G_Rule_Actions[L_i].Action_Type OF

                ACTION_SET_FLOOR_HEATING:
                    IF GVL_STATE.G_Rule_Actions[L_i].Value <= 0.0 THEN
                        GVL_COMMAND_ARBITRATION_BUFFER.B_Heating_Block := TRUE;
                        GVL_COMMAND_ARBITRATION_BUFFER.B_Boiler_Stop := TRUE;
                    END_IF;

                ACTION_SET_VENTILATION:
                    IF GVL_STATE.G_Rule_Actions[L_i].Value <= 0.0 THEN
                        GVL_COMMAND_ARBITRATION_BUFFER.B_Vent_Stop := TRUE;
                    END_IF;

            ELSE
                // Non command-level actions are handled by their own subsystem.
            END_CASE;
        END_IF;
    END_FOR;
END_IF;

IF (GVL_COMMAND_ARBITRATION_BUFFER.B_Mode = FIRE)
   AND GVL_COMMAND_POLICY_CONFIG.G_Fire_Block_Lock_Close THEN
    GVL_COMMAND_ARBITRATION_BUFFER.B_Lock_1_Close := FALSE;
    GVL_COMMAND_ARBITRATION_BUFFER.B_Lock_2_Close := FALSE;
END_IF;

IF GVL_COMMAND_POLICY_CONFIG.G_Block_Close_When_Open_Commanded THEN
    IF GVL_COMMAND_ARBITRATION_BUFFER.B_Lock_1_Open
       AND GVL_COMMAND_ARBITRATION_BUFFER.B_Lock_1_Close THEN
        GVL_COMMAND_ARBITRATION_BUFFER.B_Lock_1_Close := FALSE;
    END_IF;

    IF GVL_COMMAND_ARBITRATION_BUFFER.B_Lock_2_Open
       AND GVL_COMMAND_ARBITRATION_BUFFER.B_Lock_2_Close THEN
        GVL_COMMAND_ARBITRATION_BUFFER.B_Lock_2_Close := FALSE;
    END_IF;
END_IF;

// >>> BULK_SYNC_ANCHOR: PRG_Command_Arbitration_Phase_03_User_Rules_Conflict <<<
END_PROGRAM

(* ---- PRG_Command_Arbitration_Phase_04_Write_Shadow.st ---- *)
PROGRAM PRG_Command_Arbitration_Phase_04_Write_Shadow
// Command arbitration phase 04: single deterministic write into GVL_COMMAND_SHADOW.

GVL_COMMAND_SHADOW.G_Gas_Valve_Close := GVL_COMMAND_ARBITRATION_BUFFER.B_Gas_Valve_Close;
GVL_COMMAND_SHADOW.G_Boiler_Stop := GVL_COMMAND_ARBITRATION_BUFFER.B_Boiler_Stop;
GVL_COMMAND_SHADOW.G_Supply_100_Req := GVL_COMMAND_ARBITRATION_BUFFER.B_Supply_100_Req;
GVL_COMMAND_SHADOW.G_Supply_80_Req := GVL_COMMAND_ARBITRATION_BUFFER.B_Supply_80_Req;
GVL_COMMAND_SHADOW.G_Vent_PV3_Boost := GVL_COMMAND_ARBITRATION_BUFFER.B_Vent_PV3_Boost;
GVL_COMMAND_SHADOW.G_Exhaust_100_Req := GVL_COMMAND_ARBITRATION_BUFFER.B_Exhaust_100_Req;
GVL_COMMAND_SHADOW.G_Vent_Stop := GVL_COMMAND_ARBITRATION_BUFFER.B_Vent_Stop;
GVL_COMMAND_SHADOW.G_Vent_Block := GVL_COMMAND_ARBITRATION_BUFFER.B_Vent_Block;
GVL_COMMAND_SHADOW.G_Vent_Smoke_Exhaust := GVL_COMMAND_ARBITRATION_BUFFER.B_Vent_Smoke_Exhaust;

GVL_COMMAND_SHADOW.G_Heating_Block := GVL_COMMAND_ARBITRATION_BUFFER.B_Heating_Block;
GVL_COMMAND_SHADOW.G_Heating_Emergency_Stop := GVL_COMMAND_ARBITRATION_BUFFER.B_Heating_Emergency_Stop;
GVL_COMMAND_SHADOW.G_Heating_Gas_Safety_Stop := GVL_COMMAND_ARBITRATION_BUFFER.B_Heating_Gas_Safety_Stop;

GVL_COMMAND_SHADOW.G_Water_Block := GVL_COMMAND_ARBITRATION_BUFFER.B_Water_Block;
GVL_COMMAND_SHADOW.G_Water_Emergency_Stop := GVL_COMMAND_ARBITRATION_BUFFER.B_Water_Emergency_Stop;
GVL_COMMAND_SHADOW.G_Close_Valve_35 := GVL_COMMAND_ARBITRATION_BUFFER.B_Close_Valve_35;
GVL_COMMAND_SHADOW.G_Close_Valve_36 := GVL_COMMAND_ARBITRATION_BUFFER.B_Close_Valve_36;

GVL_COMMAND_SHADOW.G_Lock_1_Open := GVL_COMMAND_ARBITRATION_BUFFER.B_Lock_1_Open;
GVL_COMMAND_SHADOW.G_Lock_1_Close := GVL_COMMAND_ARBITRATION_BUFFER.B_Lock_1_Close;
GVL_COMMAND_SHADOW.G_Lock_2_Open := GVL_COMMAND_ARBITRATION_BUFFER.B_Lock_2_Open;
GVL_COMMAND_SHADOW.G_Lock_2_Close := GVL_COMMAND_ARBITRATION_BUFFER.B_Lock_2_Close;
GVL_COMMAND_SHADOW.G_Gate_Open := GVL_COMMAND_ARBITRATION_BUFFER.B_Gate_Open;
GVL_COMMAND_SHADOW.G_Wicket_Open := GVL_COMMAND_ARBITRATION_BUFFER.B_Wicket_Open;

// >>> BULK_SYNC_ANCHOR: PRG_Command_Arbitration_Phase_04_Write_Shadow <<<
END_PROGRAM

(* ---- PRG_Command_Verifier.st ---- *)
PROGRAM PRG_Command_Verifier
VAR
    L_i : INT;
    L_Runtime_Error : BOOL := FALSE;
    L_Runtime_Error_Code : UDINT := 0;
    L_Runtime_Error_Text : STRING(160) := '';
    L_Now_MS : UDINT;
    L_Prev_Runtime_Error : BOOL;
    L_Any_Manifold_Pump_On : BOOL;
    fbLog : FB_LogEvent;
END_VAR

L_Now_MS := GVL_STATUS.G_System_Time_MS;

// Command shadow is the current command ownership surface.
// Legacy GVL_COMMAND mismatch is intentionally not treated as a verifier fault.
GVL_COMMAND_VERIFY.Command_Mismatch_Count := 0;
GVL_COMMAND_VERIFY.Command_Match_OK := TRUE;
GVL_COMMAND_VERIFY.Command_Mismatch_Active := FALSE;

L_Runtime_Error := FALSE;
L_Runtime_Error_Code := 0;
L_Runtime_Error_Text := '';
L_Any_Manifold_Pump_On := FALSE;

IF (NOT L_Runtime_Error) AND (NOT GVL_STATUS.G_Is_Active_PLC) THEN
    FOR L_i := 1 TO GVL_CONSTANTS.C_MAX_HEATING_CIRCUITS DO
        IF GVL_IO.DO_Zone_Valves[L_i] THEN
            L_Runtime_Error := TRUE;
            L_Runtime_Error_Code := 10;
            L_Runtime_Error_Text := 'PLC inactive zone valve on';
        END_IF;
    END_FOR;
END_IF;

IF (NOT L_Runtime_Error) AND (NOT GVL_STATUS.G_Is_Active_PLC) THEN
    FOR L_i := 1 TO GVL_CONSTANTS.C_MAX_MANIFOLDS DO
        IF GVL_IO.DO_Manifold_Pumps[L_i] THEN
            L_Runtime_Error := TRUE;
            L_Runtime_Error_Code := 11;
            L_Runtime_Error_Text := 'PLC inactive pump on';
        END_IF;
    END_FOR;
END_IF;

IF (NOT L_Runtime_Error) AND (GVL_SAFETY_SHUTDOWN.G_Safety_Mode = GAS) AND (NOT GVL_IO.DO_Gas_Valve_Close) THEN
    L_Runtime_Error := TRUE;
    L_Runtime_Error_Code := 1;
    L_Runtime_Error_Text := 'Gas valve not closed';
END_IF;

IF (NOT L_Runtime_Error) AND (GVL_SAFETY_SHUTDOWN.G_Safety_Mode = GAS) THEN
    IF (GVL_IO.AO_Supply_Fans[1] = 0) AND (GVL_IO.AO_Exhaust_Fans[1] = 0) THEN
        L_Runtime_Error := TRUE;
        L_Runtime_Error_Code := 3;
        L_Runtime_Error_Text := 'Gas ventilation inactive';
    END_IF;
END_IF;

IF (NOT L_Runtime_Error) AND (GVL_SAFETY_SHUTDOWN.G_Safety_Mode = FIRE) THEN
    FOR L_i := 1 TO GVL_CONSTANTS.C_MAX_EXHAUST_FANS DO
        IF GVL_IO.AO_Exhaust_Fans[L_i] = 0 THEN
            L_Runtime_Error := TRUE;
            L_Runtime_Error_Code := 2;
            L_Runtime_Error_Text := 'Smoke exhaust not active';
        END_IF;
    END_FOR;
END_IF;

IF (NOT L_Runtime_Error) AND (GVL_SAFETY_SHUTDOWN.G_Safety_Mode = FIRE) THEN
    FOR L_i := 1 TO GVL_CONSTANTS.C_MAX_SUPPLY_FANS DO
        IF GVL_IO.AO_Supply_Fans[L_i] <> 0 THEN
            L_Runtime_Error := TRUE;
            L_Runtime_Error_Code := 4;
            L_Runtime_Error_Text := 'Supply fan active in fire';
        END_IF;
    END_FOR;
END_IF;

IF (NOT L_Runtime_Error) AND (GVL_SAFETY_SHUTDOWN.G_Safety_Mode = WATER_LEAK) THEN
    IF GVL_COMMAND_SHADOW.G_Close_Valve_35 AND (NOT GVL_IO.DO_Water_Valve_35_Close) THEN
        L_Runtime_Error := TRUE;
        L_Runtime_Error_Code := 5;
        L_Runtime_Error_Text := 'Water valve 35 not closed';
    ELSIF GVL_COMMAND_SHADOW.G_Close_Valve_36 AND (NOT GVL_IO.DO_Water_Valve_36_Close) THEN
        L_Runtime_Error := TRUE;
        L_Runtime_Error_Code := 6;
        L_Runtime_Error_Text := 'Water valve 36 not closed';
    END_IF;
END_IF;

IF (NOT L_Runtime_Error) AND GVL_STATE.G_Safety_Freeze_Risk THEN
    FOR L_i := 1 TO GVL_CONSTANTS.C_MAX_MANIFOLDS DO
        IF GVL_IO.DO_Manifold_Pumps[L_i] THEN
            L_Any_Manifold_Pump_On := TRUE;
        END_IF;
    END_FOR;

    IF (NOT L_Any_Manifold_Pump_On) AND (NOT GVL_IO.DO_Backup_Circulation_Pump) THEN
        L_Runtime_Error := TRUE;
        L_Runtime_Error_Code := 7;
        L_Runtime_Error_Text := 'Freeze circulation inactive';
    END_IF;
END_IF;

IF (NOT L_Runtime_Error) AND GVL_STATE.G_Safety_Freeze_Risk AND GVL_COMMAND_SHADOW.G_Heating_Gas_Safety_Stop THEN
    IF GVL_IO.DO_DHW_Heating_Pump THEN
        L_Runtime_Error := TRUE;
        L_Runtime_Error_Code := 8;
        L_Runtime_Error_Text := 'DHW heating active during gas freeze';
    END_IF;
END_IF;

IF L_Runtime_Error THEN
    GVL_COMMAND_VERIFY.Runtime_Sanity_OK := FALSE;
    GVL_COMMAND_VERIFY.Runtime_Last_Error_Code := L_Runtime_Error_Code;
    GVL_COMMAND_VERIFY.Runtime_Last_Error_Text := L_Runtime_Error_Text;
    GVL_COMMAND_VERIFY.Runtime_Last_Error_Time_MS := L_Now_MS;

    IF NOT L_Prev_Runtime_Error THEN
        GVL_COMMAND_VERIFY.Runtime_Sanity_Error_Count := GVL_COMMAND_VERIFY.Runtime_Sanity_Error_Count + 1;
        fbLog(
            VI_Event_Type := 1001,
            VI_Timestamp := L_Now_MS,
            VI_Param1 := L_Runtime_Error_Code,
            VI_Param2 := GVL_COMMAND_VERIFY.Runtime_Sanity_Error_Count
        );
    END_IF;
ELSE
    GVL_COMMAND_VERIFY.Runtime_Sanity_OK := TRUE;
END_IF;

L_Prev_Runtime_Error := L_Runtime_Error;

END_PROGRAM

(* ---- PRG_Compliance_Federation_Governor.st ---- *)
PROGRAM PRG_Compliance_Federation_Governor
VAR
    L_Now_MS : UDINT;
    L_Compliance_Valid : BOOL := TRUE;
    L_Error_Code : UDINT := 0;
    L_Error_Text : STRING(160) := '';
END_VAR

L_Now_MS := GVL_STATUS.G_System_Time_MS;
L_Compliance_Valid := TRUE;
L_Error_Code := 0;
L_Error_Text := '';

// Fail-safe defaults.
GVL_COMPLIANCE_FEDERATION_FABRIC.Compliance_Federation_Valid := FALSE;
GVL_COMPLIANCE_FEDERATION_FABRIC.Compliance_Federation_Granted := FALSE;
GVL_COMPLIANCE_FEDERATION_FABRIC.Compliance_Federation_Quarantine_Active := TRUE;

GVL_COMPLIANCE_FEDERATION_FABRIC.Regulatory_Semantics_Coherent := FALSE;
GVL_COMPLIANCE_FEDERATION_FABRIC.Certification_Boundary_Valid := FALSE;
GVL_COMPLIANCE_FEDERATION_FABRIC.Regional_Safety_Envelope_Aligned := FALSE;
GVL_COMPLIANCE_FEDERATION_FABRIC.Governance_Trust_Boundary_Stable := FALSE;
GVL_COMPLIANCE_FEDERATION_FABRIC.Policy_Compliance_Coherent := FALSE;

// Semantic federation required.
IF NOT GVL_SEMANTIC_FEDERATION_FABRIC.Semantic_Federation_Granted THEN
    L_Compliance_Valid := FALSE;
    L_Error_Code := 42000;
    L_Error_Text := 'Semantic federation authority not granted';
END_IF;

// Regulatory semantic split-brain detectors.
IF GVL_COMPLIANCE_FEDERATION_FABRIC.CrossJurisdiction_Semantic_Drift_Detected THEN
    L_Compliance_Valid := FALSE;
    L_Error_Code := 42001;
    L_Error_Text := 'Cross-jurisdiction semantic drift detected';
END_IF;

IF GVL_COMPLIANCE_FEDERATION_FABRIC.Certification_Boundary_Violation_Detected THEN
    L_Compliance_Valid := FALSE;
    L_Error_Code := 42002;
    L_Error_Text := 'Certification boundary violation detected';
END_IF;

IF GVL_COMPLIANCE_FEDERATION_FABRIC.Policy_Compliance_Divergence_Detected THEN
    L_Compliance_Valid := FALSE;
    L_Error_Code := 42003;
    L_Error_Text := 'Policy compliance divergence detected';
END_IF;

IF GVL_COMPLIANCE_FEDERATION_FABRIC.Regional_Safety_Envelope_Mismatch_Detected THEN
    L_Compliance_Valid := FALSE;
    L_Error_Code := 42004;
    L_Error_Text := 'Regional safety envelope mismatch detected';
END_IF;

IF GVL_COMPLIANCE_FEDERATION_FABRIC.Regulatory_Trust_Corruption_Detected THEN
    L_Compliance_Valid := FALSE;
    L_Error_Code := 42005;
    L_Error_Text := 'Regulatory trust corruption detected';
END_IF;

IF GVL_COMPLIANCE_FEDERATION_FABRIC.Governance_Authority_Leakage_Detected THEN
    L_Compliance_Valid := FALSE;
    L_Error_Code := 42006;
    L_Error_Text := 'Governance authority leakage detected';
END_IF;

// Compliance federation validation.
IF L_Compliance_Valid
AND NOT GVL_COMPLIANCE_FEDERATION_FABRIC.CrossJurisdiction_Authority_Aligned THEN
    L_Compliance_Valid := FALSE;
    L_Error_Code := 42010;
    L_Error_Text := 'Cross-jurisdiction authority alignment invalid';
END_IF;

IF L_Compliance_Valid
AND NOT GVL_COMPLIANCE_FEDERATION_FABRIC.Compliance_Runtime_Projection_Stable THEN
    L_Compliance_Valid := FALSE;
    L_Error_Code := 42011;
    L_Error_Text := 'Compliance runtime projection unstable';
END_IF;

IF L_Compliance_Valid
AND NOT GVL_COMPLIANCE_FEDERATION_FABRIC.External_Governance_Interpretation_Valid THEN
    L_Compliance_Valid := FALSE;
    L_Error_Code := 42012;
    L_Error_Text := 'External governance interpretation invalid';
END_IF;

IF L_Compliance_Valid
AND NOT GVL_COMPLIANCE_FEDERATION_FABRIC.Certified_Operational_Semantics_Valid THEN
    L_Compliance_Valid := FALSE;
    L_Error_Code := 42013;
    L_Error_Text := 'Certified operational semantics invalid';
END_IF;

IF L_Compliance_Valid THEN
    GVL_COMPLIANCE_FEDERATION_FABRIC.Compliance_Federation_Valid := TRUE;
    GVL_COMPLIANCE_FEDERATION_FABRIC.Compliance_Federation_Granted := TRUE;
    GVL_COMPLIANCE_FEDERATION_FABRIC.Compliance_Federation_Quarantine_Active := FALSE;

    GVL_COMPLIANCE_FEDERATION_FABRIC.Regulatory_Semantics_Coherent := TRUE;
    GVL_COMPLIANCE_FEDERATION_FABRIC.Certification_Boundary_Valid := TRUE;
    GVL_COMPLIANCE_FEDERATION_FABRIC.Regional_Safety_Envelope_Aligned := TRUE;
    GVL_COMPLIANCE_FEDERATION_FABRIC.Governance_Trust_Boundary_Stable := TRUE;
    GVL_COMPLIANCE_FEDERATION_FABRIC.Policy_Compliance_Coherent := TRUE;

    GVL_COMPLIANCE_FEDERATION_FABRIC.Compliance_Federation_Epoch :=
        GVL_SEMANTIC_FEDERATION_FABRIC.Semantic_Federation_Epoch;

    GVL_COMPLIANCE_FEDERATION_FABRIC.Compliance_Federation_Epoch_Coherent := TRUE;

    GVL_COMPLIANCE_FEDERATION_FABRIC.Compliance_Federation_Last_Update_MS :=
        L_Now_MS;

    GVL_COMPLIANCE_FEDERATION_FABRIC.Compliance_Federation_Lease_Expired := FALSE;

    GVL_COMPLIANCE_FEDERATION_FABRIC.Compliance_Federation_Last_Error_Code := 0;
    GVL_COMPLIANCE_FEDERATION_FABRIC.Compliance_Federation_Last_Error_Text := '';
ELSE
    GVL_COMPLIANCE_FEDERATION_FABRIC.Compliance_Federation_Valid := FALSE;
    GVL_COMPLIANCE_FEDERATION_FABRIC.Compliance_Federation_Granted := FALSE;
    GVL_COMPLIANCE_FEDERATION_FABRIC.Compliance_Federation_Quarantine_Active := TRUE;

    GVL_COMPLIANCE_FEDERATION_FABRIC.Compliance_Federation_Lease_Expired := TRUE;

    GVL_COMPLIANCE_FEDERATION_FABRIC.Compliance_Federation_Last_Error_Code :=
        L_Error_Code;

    GVL_COMPLIANCE_FEDERATION_FABRIC.Compliance_Federation_Last_Error_Text :=
        L_Error_Text;

    GVL_COMPLIANCE_FEDERATION_FABRIC.Compliance_Federation_Invalidation_Count :=
        GVL_COMPLIANCE_FEDERATION_FABRIC.Compliance_Federation_Invalidation_Count + 1;
END_IF;

END_PROGRAM

(* ---- PRG_Config_Manager.st ---- *)
PROGRAM PRG_Config_Manager
VAR
    L_Error : BOOL;
    L_Staged_Error : BOOL;
    L_Index : INT;
END_VAR

L_Error := FALSE;
L_Staged_Error := FALSE;
GVL_CONFIG_VALIDATION.G_Config_Auto_Corrected := FALSE;
GVL_CONFIG_VALIDATION.G_Config_Reset_To_Default_Done := FALSE;
GVL_CONFIG_CONTROL.G_Apply_Done := FALSE;
GVL_CONFIG_CONTROL.G_Rollback_Done := FALSE;

// ===== SIZE VALIDATION =====
IF GVL_SYSTEM_SIZE_CONFIG.G_Active_Heating_Circuits < 1 OR GVL_SYSTEM_SIZE_CONFIG.G_Active_Heating_Circuits > GVL_CONSTANTS.C_MAX_HEATING_CIRCUITS THEN
    GVL_SYSTEM_SIZE_CONFIG.G_Active_Heating_Circuits := GVL_CONSTANTS.C_MAX_HEATING_CIRCUITS;
    L_Error := TRUE;
END_IF;

IF GVL_SYSTEM_SIZE_CONFIG.G_Active_Water_Zones < 1 OR GVL_SYSTEM_SIZE_CONFIG.G_Active_Water_Zones > GVL_CONSTANTS.C_MAX_WATER_ZONES THEN
    GVL_SYSTEM_SIZE_CONFIG.G_Active_Water_Zones := GVL_CONSTANTS.C_MAX_WATER_ZONES;
    L_Error := TRUE;
END_IF;

IF GVL_SYSTEM_SIZE_CONFIG.G_Active_Light_Zones < 1 OR GVL_SYSTEM_SIZE_CONFIG.G_Active_Light_Zones > GVL_CONSTANTS.C_MAX_LIGHT_ZONES THEN
    GVL_SYSTEM_SIZE_CONFIG.G_Active_Light_Zones := GVL_CONSTANTS.C_MAX_LIGHT_ZONES;
    L_Error := TRUE;
END_IF;

// ===== EXISTING ACTIVE VALIDATION =====
IF GVL_INPUT_VALIDATION_CONFIG.G_Reputation_Learning_Rate < 0.0 OR GVL_INPUT_VALIDATION_CONFIG.G_Reputation_Learning_Rate > 1.0 THEN
    GVL_INPUT_VALIDATION_CONFIG.G_Reputation_Learning_Rate := 0.05;
    L_Error := TRUE;
END_IF;

// ===== APPLY STAGED CONFIG =====
IF GVL_CONFIG_CONTROL.G_Apply_Request AND GVL_CONFIG_CONTROL.G_Apply_Confirm THEN
    L_Staged_Error := FALSE;

    IF (GVL_CONFIG_CONTROL.STG_Reputation_Learning_Rate < 0.0) OR (GVL_CONFIG_CONTROL.STG_Reputation_Learning_Rate > 1.0) THEN
        L_Staged_Error := TRUE;
    END_IF;

    IF (GVL_CONFIG_CONTROL.STG_Reputation_Recovery_Decay < 0.0) OR (GVL_CONFIG_CONTROL.STG_Reputation_Recovery_Decay > 1.0) THEN
        L_Staged_Error := TRUE;
    END_IF;

    IF (GVL_CONFIG_CONTROL.STG_Min_Sensor_Confidence < 0.0) OR (GVL_CONFIG_CONTROL.STG_Min_Sensor_Confidence > 1.0) THEN
        L_Staged_Error := TRUE;
    END_IF;

    IF (GVL_CONFIG_CONTROL.STG_Bad_Spike_Confidence < 0.0) OR (GVL_CONFIG_CONTROL.STG_Bad_Spike_Confidence > 1.0) THEN
        L_Staged_Error := TRUE;
    END_IF;

    IF (GVL_CONFIG_CONTROL.STG_Default_Confidence < 0.0) OR (GVL_CONFIG_CONTROL.STG_Default_Confidence > 1.0) THEN
        L_Staged_Error := TRUE;
    END_IF;

    IF (GVL_CONFIG_CONTROL.STG_Night_Start_Hour < 0) OR (GVL_CONFIG_CONTROL.STG_Night_Start_Hour > 23) THEN
        L_Staged_Error := TRUE;
    END_IF;

    IF (GVL_CONFIG_CONTROL.STG_Night_End_Hour < 0) OR (GVL_CONFIG_CONTROL.STG_Night_End_Hour > 23) THEN
        L_Staged_Error := TRUE;
    END_IF;

    IF (GVL_CONFIG_CONTROL.STG_VentBoost_Humidity_Threshold < 0.0) OR (GVL_CONFIG_CONTROL.STG_VentBoost_Humidity_Threshold > 100.0) THEN
        L_Staged_Error := TRUE;
    END_IF;

    IF GVL_CONFIG_CONTROL.STG_Stabilization_Delay_MS < 1000 THEN
        L_Staged_Error := TRUE;
    END_IF;

    IF NOT GVL_CONFIG_SIMULATION.G_Simulation_Result_OK THEN
        L_Staged_Error := TRUE;
    END_IF;

    IF L_Staged_Error THEN
        L_Index := GVL_CONFIG_HISTORY.G_History_Index;
        GVL_CONFIG_HISTORY.G_History_Version[L_Index] := GVL_CONFIG_CONTROL.G_Config_Version;
        GVL_CONFIG_HISTORY.G_History_Time_MS[L_Index] := GVL_TIME_SERVICE.G_Now_MS;
        GVL_CONFIG_HISTORY.G_History_Action[L_Index] := 'APPLY_REJECTED';
        GVL_CONFIG_HISTORY.G_Last_Action_Text := 'CONFIG APPLY REJECTED';

        L_Index := L_Index + 1;
        IF L_Index > 5 THEN L_Index := 1; END_IF;
        GVL_CONFIG_HISTORY.G_History_Index := L_Index;

        GVL_CONFIG_VALIDATION.G_Config_Control_Error_Text := 'STAGED CONFIG INVALID';
    ELSE
        // Backup current active values before applying staged values.
        GVL_CONFIG_CONTROL.BCK_Reputation_Learning_Rate := GVL_INPUT_VALIDATION_CONFIG.G_Reputation_Learning_Rate;
        GVL_CONFIG_CONTROL.BCK_Reputation_Recovery_Decay := GVL_INPUT_VALIDATION_CONFIG.G_Reputation_Recovery_Decay;
        GVL_CONFIG_CONTROL.BCK_Min_Sensor_Confidence := GVL_INPUT_VALIDATION_CONFIG.G_Min_Sensor_Confidence;
        GVL_CONFIG_CONTROL.BCK_Bad_Spike_Confidence := GVL_INPUT_VALIDATION_CONFIG.G_Bad_Spike_Confidence;
        GVL_CONFIG_CONTROL.BCK_Default_Confidence := GVL_INPUT_VALIDATION_CONFIG.G_Default_Confidence;

        GVL_CONFIG_CONTROL.BCK_Night_Start_Hour := GVL_SCENARIO_CONFIG.G_Night_Start_Hour;
        GVL_CONFIG_CONTROL.BCK_Night_End_Hour := GVL_SCENARIO_CONFIG.G_Night_End_Hour;
        GVL_CONFIG_CONTROL.BCK_VentBoost_Humidity_Threshold := GVL_SCENARIO_CONFIG.G_VentBoost_Humidity_Threshold;

        GVL_CONFIG_CONTROL.BCK_Stabilization_Delay_MS := GVL_SAFETY_RECOVERY_CONFIG.G_Stabilization_Delay_MS;

        GVL_CONFIG_CONTROL.BCK_PLC_Inactive_Close_Gas := GVL_COMMAND_POLICY_CONFIG.G_PLC_Inactive_Close_Gas;
        GVL_CONFIG_CONTROL.BCK_PLC_Inactive_Stop_Boiler := GVL_COMMAND_POLICY_CONFIG.G_PLC_Inactive_Stop_Boiler;
        GVL_CONFIG_CONTROL.BCK_PLC_Inactive_Block_Heating := GVL_COMMAND_POLICY_CONFIG.G_PLC_Inactive_Block_Heating;
        GVL_CONFIG_CONTROL.BCK_PLC_Inactive_Stop_Vent := GVL_COMMAND_POLICY_CONFIG.G_PLC_Inactive_Stop_Vent;
        GVL_CONFIG_CONTROL.BCK_PLC_Inactive_Block_Water := GVL_COMMAND_POLICY_CONFIG.G_PLC_Inactive_Block_Water;

        // Apply staged input config.
        GVL_INPUT_VALIDATION_CONFIG.G_Reputation_Learning_Rate := GVL_CONFIG_CONTROL.STG_Reputation_Learning_Rate;
        GVL_INPUT_VALIDATION_CONFIG.G_Reputation_Recovery_Decay := GVL_CONFIG_CONTROL.STG_Reputation_Recovery_Decay;
        GVL_INPUT_VALIDATION_CONFIG.G_Min_Sensor_Confidence := GVL_CONFIG_CONTROL.STG_Min_Sensor_Confidence;
        GVL_INPUT_VALIDATION_CONFIG.G_Bad_Spike_Confidence := GVL_CONFIG_CONTROL.STG_Bad_Spike_Confidence;
        GVL_INPUT_VALIDATION_CONFIG.G_Default_Confidence := GVL_CONFIG_CONTROL.STG_Default_Confidence;

        // Apply staged scenario config.
        GVL_SCENARIO_CONFIG.G_Night_Start_Hour := GVL_CONFIG_CONTROL.STG_Night_Start_Hour;
        GVL_SCENARIO_CONFIG.G_Night_End_Hour := GVL_CONFIG_CONTROL.STG_Night_End_Hour;
        GVL_SCENARIO_CONFIG.G_VentBoost_Humidity_Threshold := GVL_CONFIG_CONTROL.STG_VentBoost_Humidity_Threshold;

        // Apply staged recovery config.
        GVL_SAFETY_RECOVERY_CONFIG.G_Stabilization_Delay_MS := GVL_CONFIG_CONTROL.STG_Stabilization_Delay_MS;

        // Apply staged command-policy critical config.
        GVL_COMMAND_POLICY_CONFIG.G_PLC_Inactive_Close_Gas := GVL_CONFIG_CONTROL.STG_PLC_Inactive_Close_Gas;
        GVL_COMMAND_POLICY_CONFIG.G_PLC_Inactive_Stop_Boiler := GVL_CONFIG_CONTROL.STG_PLC_Inactive_Stop_Boiler;
        GVL_COMMAND_POLICY_CONFIG.G_PLC_Inactive_Block_Heating := GVL_CONFIG_CONTROL.STG_PLC_Inactive_Block_Heating;
        GVL_COMMAND_POLICY_CONFIG.G_PLC_Inactive_Stop_Vent := GVL_CONFIG_CONTROL.STG_PLC_Inactive_Stop_Vent;
        GVL_COMMAND_POLICY_CONFIG.G_PLC_Inactive_Block_Water := GVL_CONFIG_CONTROL.STG_PLC_Inactive_Block_Water;

        GVL_CONFIG_CONTROL.G_Config_Version := GVL_CONFIG_CONTROL.G_Config_Version + 1;
        GVL_CONFIG_CONTROL.G_Last_Good_Version := GVL_CONFIG_CONTROL.G_Config_Version;
        GVL_CONFIG_CONTROL.G_Backup_Valid := TRUE;
        GVL_CONFIG_CONTROL.G_Apply_Done := TRUE;
        GVL_CONFIG_VALIDATION.G_Config_Control_Error_Text := '';

        L_Index := GVL_CONFIG_HISTORY.G_History_Index;
        GVL_CONFIG_HISTORY.G_History_Version[L_Index] := GVL_CONFIG_CONTROL.G_Config_Version;
        GVL_CONFIG_HISTORY.G_History_Time_MS[L_Index] := GVL_TIME_SERVICE.G_Now_MS;
        GVL_CONFIG_HISTORY.G_History_Action[L_Index] := 'APPLY';
        GVL_CONFIG_HISTORY.G_Last_Action_Text := 'CONFIG APPLY';

        L_Index := L_Index + 1;
        IF L_Index > 5 THEN L_Index := 1; END_IF;
        GVL_CONFIG_HISTORY.G_History_Index := L_Index;
    END_IF;

    GVL_CONFIG_CONTROL.G_Apply_Request := FALSE;
    GVL_CONFIG_CONTROL.G_Apply_Confirm := FALSE;
END_IF;

// ===== RESET CONTROLLED CONFIG TO DEFAULTS =====
IF GVL_CONFIG_CONTROL.G_Reset_Default_Request AND GVL_CONFIG_CONTROL.G_Reset_Default_Confirm THEN
    // Backup current active values before resetting controlled config defaults.
    GVL_CONFIG_CONTROL.BCK_Reputation_Learning_Rate := GVL_INPUT_VALIDATION_CONFIG.G_Reputation_Learning_Rate;
    GVL_CONFIG_CONTROL.BCK_Reputation_Recovery_Decay := GVL_INPUT_VALIDATION_CONFIG.G_Reputation_Recovery_Decay;
    GVL_CONFIG_CONTROL.BCK_Min_Sensor_Confidence := GVL_INPUT_VALIDATION_CONFIG.G_Min_Sensor_Confidence;
    GVL_CONFIG_CONTROL.BCK_Bad_Spike_Confidence := GVL_INPUT_VALIDATION_CONFIG.G_Bad_Spike_Confidence;
    GVL_CONFIG_CONTROL.BCK_Default_Confidence := GVL_INPUT_VALIDATION_CONFIG.G_Default_Confidence;

    GVL_CONFIG_CONTROL.BCK_Night_Start_Hour := GVL_SCENARIO_CONFIG.G_Night_Start_Hour;
    GVL_CONFIG_CONTROL.BCK_Night_End_Hour := GVL_SCENARIO_CONFIG.G_Night_End_Hour;
    GVL_CONFIG_CONTROL.BCK_VentBoost_Humidity_Threshold := GVL_SCENARIO_CONFIG.G_VentBoost_Humidity_Threshold;

    GVL_CONFIG_CONTROL.BCK_Stabilization_Delay_MS := GVL_SAFETY_RECOVERY_CONFIG.G_Stabilization_Delay_MS;

    GVL_CONFIG_CONTROL.BCK_PLC_Inactive_Close_Gas := GVL_COMMAND_POLICY_CONFIG.G_PLC_Inactive_Close_Gas;
    GVL_CONFIG_CONTROL.BCK_PLC_Inactive_Stop_Boiler := GVL_COMMAND_POLICY_CONFIG.G_PLC_Inactive_Stop_Boiler;
    GVL_CONFIG_CONTROL.BCK_PLC_Inactive_Block_Heating := GVL_COMMAND_POLICY_CONFIG.G_PLC_Inactive_Block_Heating;
    GVL_CONFIG_CONTROL.BCK_PLC_Inactive_Stop_Vent := GVL_COMMAND_POLICY_CONFIG.G_PLC_Inactive_Stop_Vent;
    GVL_CONFIG_CONTROL.BCK_PLC_Inactive_Block_Water := GVL_COMMAND_POLICY_CONFIG.G_PLC_Inactive_Block_Water;

    // Reset staged and active controlled config values to conservative defaults.
    GVL_CONFIG_CONTROL.STG_Reputation_Learning_Rate := 0.05;
    GVL_CONFIG_CONTROL.STG_Reputation_Recovery_Decay := 0.01;
    GVL_CONFIG_CONTROL.STG_Min_Sensor_Confidence := 0.1;
    GVL_CONFIG_CONTROL.STG_Bad_Spike_Confidence := 0.3;
    GVL_CONFIG_CONTROL.STG_Default_Confidence := 1.0;

    GVL_INPUT_VALIDATION_CONFIG.G_Reputation_Learning_Rate := 0.05;
    GVL_INPUT_VALIDATION_CONFIG.G_Reputation_Recovery_Decay := 0.01;
    GVL_INPUT_VALIDATION_CONFIG.G_Min_Sensor_Confidence := 0.1;
    GVL_INPUT_VALIDATION_CONFIG.G_Bad_Spike_Confidence := 0.3;
    GVL_INPUT_VALIDATION_CONFIG.G_Default_Confidence := 1.0;

    GVL_CONFIG_CONTROL.STG_Night_Start_Hour := 22;
    GVL_CONFIG_CONTROL.STG_Night_End_Hour := 6;
    GVL_CONFIG_CONTROL.STG_VentBoost_Humidity_Threshold := 65.0;

    GVL_SCENARIO_CONFIG.G_Night_Start_Hour := 22;
    GVL_SCENARIO_CONFIG.G_Night_End_Hour := 6;
    GVL_SCENARIO_CONFIG.G_VentBoost_Humidity_Threshold := 65.0;

    GVL_CONFIG_CONTROL.STG_Stabilization_Delay_MS := 5000;
    GVL_SAFETY_RECOVERY_CONFIG.G_Stabilization_Delay_MS := 5000;

    GVL_CONFIG_CONTROL.STG_PLC_Inactive_Close_Gas := TRUE;
    GVL_CONFIG_CONTROL.STG_PLC_Inactive_Stop_Boiler := TRUE;
    GVL_CONFIG_CONTROL.STG_PLC_Inactive_Block_Heating := TRUE;
    GVL_CONFIG_CONTROL.STG_PLC_Inactive_Stop_Vent := TRUE;
    GVL_CONFIG_CONTROL.STG_PLC_Inactive_Block_Water := TRUE;

    GVL_COMMAND_POLICY_CONFIG.G_PLC_Inactive_Close_Gas := TRUE;
    GVL_COMMAND_POLICY_CONFIG.G_PLC_Inactive_Stop_Boiler := TRUE;
    GVL_COMMAND_POLICY_CONFIG.G_PLC_Inactive_Block_Heating := TRUE;
    GVL_COMMAND_POLICY_CONFIG.G_PLC_Inactive_Stop_Vent := TRUE;
    GVL_COMMAND_POLICY_CONFIG.G_PLC_Inactive_Block_Water := TRUE;

    GVL_CONFIG_CONTROL.G_Config_Version := GVL_CONFIG_CONTROL.G_Config_Version + 1;
    GVL_CONFIG_CONTROL.G_Last_Good_Version := GVL_CONFIG_CONTROL.G_Config_Version;
    GVL_CONFIG_CONTROL.G_Backup_Valid := TRUE;
    GVL_CONFIG_VALIDATION.G_Config_Reset_To_Default_Done := TRUE;
    GVL_CONFIG_VALIDATION.G_Config_Control_Error_Text := '';

    L_Index := GVL_CONFIG_HISTORY.G_History_Index;
    GVL_CONFIG_HISTORY.G_History_Version[L_Index] := GVL_CONFIG_CONTROL.G_Config_Version;
    GVL_CONFIG_HISTORY.G_History_Time_MS[L_Index] := GVL_TIME_SERVICE.G_Now_MS;
    GVL_CONFIG_HISTORY.G_History_Action[L_Index] := 'RESET_DEFAULT';
    GVL_CONFIG_HISTORY.G_Last_Action_Text := 'CONFIG RESET DEFAULT';

    L_Index := L_Index + 1;
    IF L_Index > 5 THEN L_Index := 1; END_IF;
    GVL_CONFIG_HISTORY.G_History_Index := L_Index;

    GVL_CONFIG_CONTROL.G_Reset_Default_Request := FALSE;
    GVL_CONFIG_CONTROL.G_Reset_Default_Confirm := FALSE;
END_IF;

// ===== ROLLBACK TO LAST BACKUP =====
IF GVL_CONFIG_CONTROL.G_Rollback_Request AND GVL_CONFIG_CONTROL.G_Rollback_Confirm THEN
    IF GVL_CONFIG_CONTROL.G_Backup_Valid THEN
        GVL_INPUT_VALIDATION_CONFIG.G_Reputation_Learning_Rate := GVL_CONFIG_CONTROL.BCK_Reputation_Learning_Rate;
        GVL_INPUT_VALIDATION_CONFIG.G_Reputation_Recovery_Decay := GVL_CONFIG_CONTROL.BCK_Reputation_Recovery_Decay;
        GVL_INPUT_VALIDATION_CONFIG.G_Min_Sensor_Confidence := GVL_CONFIG_CONTROL.BCK_Min_Sensor_Confidence;
        GVL_INPUT_VALIDATION_CONFIG.G_Bad_Spike_Confidence := GVL_CONFIG_CONTROL.BCK_Bad_Spike_Confidence;
        GVL_INPUT_VALIDATION_CONFIG.G_Default_Confidence := GVL_CONFIG_CONTROL.BCK_Default_Confidence;

        GVL_SCENARIO_CONFIG.G_Night_Start_Hour := GVL_CONFIG_CONTROL.BCK_Night_Start_Hour;
        GVL_SCENARIO_CONFIG.G_Night_End_Hour := GVL_CONFIG_CONTROL.BCK_Night_End_Hour;
        GVL_SCENARIO_CONFIG.G_VentBoost_Humidity_Threshold := GVL_CONFIG_CONTROL.BCK_VentBoost_Humidity_Threshold;

        GVL_SAFETY_RECOVERY_CONFIG.G_Stabilization_Delay_MS := GVL_CONFIG_CONTROL.BCK_Stabilization_Delay_MS;

        GVL_COMMAND_POLICY_CONFIG.G_PLC_Inactive_Close_Gas := GVL_CONFIG_CONTROL.BCK_PLC_Inactive_Close_Gas;
        GVL_COMMAND_POLICY_CONFIG.G_PLC_Inactive_Stop_Boiler := GVL_CONFIG_CONTROL.BCK_PLC_Inactive_Stop_Boiler;
        GVL_COMMAND_POLICY_CONFIG.G_PLC_Inactive_Block_Heating := GVL_CONFIG_CONTROL.BCK_PLC_Inactive_Block_Heating;
        GVL_COMMAND_POLICY_CONFIG.G_PLC_Inactive_Stop_Vent := GVL_CONFIG_CONTROL.BCK_PLC_Inactive_Stop_Vent;
        GVL_COMMAND_POLICY_CONFIG.G_PLC_Inactive_Block_Water := GVL_CONFIG_CONTROL.BCK_PLC_Inactive_Block_Water;

        GVL_CONFIG_CONTROL.G_Config_Version := GVL_CONFIG_CONTROL.G_Config_Version + 1;
        GVL_CONFIG_CONTROL.G_Rollback_Done := TRUE;
        GVL_CONFIG_VALIDATION.G_Config_Control_Error_Text := '';

        L_Index := GVL_CONFIG_HISTORY.G_History_Index;
        GVL_CONFIG_HISTORY.G_History_Version[L_Index] := GVL_CONFIG_CONTROL.G_Config_Version;
        GVL_CONFIG_HISTORY.G_History_Time_MS[L_Index] := GVL_TIME_SERVICE.G_Now_MS;
        GVL_CONFIG_HISTORY.G_History_Action[L_Index] := 'ROLLBACK';
        GVL_CONFIG_HISTORY.G_Last_Action_Text := 'CONFIG ROLLBACK';

        L_Index := L_Index + 1;
        IF L_Index > 5 THEN L_Index := 1; END_IF;
        GVL_CONFIG_HISTORY.G_History_Index := L_Index;
    ELSE
        GVL_CONFIG_HISTORY.G_Last_Action_Text := 'CONFIG ROLLBACK REJECTED - NO BACKUP';
        GVL_CONFIG_VALIDATION.G_Config_Control_Error_Text := 'ROLLBACK REJECTED - NO BACKUP';
    END_IF;

    GVL_CONFIG_CONTROL.G_Rollback_Request := FALSE;
    GVL_CONFIG_CONTROL.G_Rollback_Confirm := FALSE;
END_IF;

GVL_CONFIG_VALIDATION.G_Config_Valid := NOT L_Error;
GVL_CONFIG_VALIDATION.G_Config_Last_Update_MS := GVL_TIME_SERVICE.G_Now_MS;

// >>> BULK_SYNC_ANCHOR: PRG_Config_Manager <<<
END_PROGRAM
